     //Waga 1                                                   
	iWeight1State										:INT;						// Stan
	sWeight1State										:STRING;					// Stan
	bWeight1DoWeighting									:BOOL;						// Ważenie
	bWeight1Tare										:BOOL;						// Taruj
	lrWeight1Measured									:LREAL;						// Waga [g]
	lrWeight1Mass										:LREAL;						// Waga masy [g] (na ekranie głównym)
	//Waga 2
	iWeight2State										:INT;						// Stan
	sWeight2State										:STRING;					// Stan
	bWeight2DoWeighting									:BOOL;						// Ważenie
	bWeight2Tare										:BOOL;						// Taruj
	lrWeight2Measured									:LREAL;						// Waga [g]
	lrWeight2Mass										:LREAL;						// Waga masy [g] (na ekranie głównym)
	//Waga 3
	iWeight3State										:INT;						// Stan
	sWeight3State										:STRING;					// Stan
	bWeight3DoWeighting									:BOOL;						// Ważenie
	bWeight3Tare										:BOOL;						// Taruj
	lrWeight3Measured									:LREAL;						// Waga [g]
	lrWeight3Mass										:LREAL;						// Waga masy [g] (na ekranie głównym)
	//Waga 4
	iWeight4State										:INT;						// Stan
	sWeight4State										:STRING;					// Stan
	bWeight4DoWeighting									:BOOL;						// Ważenie
	bWeight4Tare										:BOOL;						// Taruj
	lrWeight4Measured									:LREAL;						// Waga [g]
	lrWeight4Mass										:LREAL;						// Waga masy [g] (na ekranie głównym)
	//Waga 5	
	iWeight5State										:INT;						// Stan
	sWeight5State										:STRING;					// Stan
	bWeight5DoWeighting									:BOOL;						// Ważenie
	bWeight5Tare										:BOOL;						// Taruj
	lrWeight5Measured									:LREAL;						// Waga [g]
	lrWeight5Mass										:LREAL;						// Waga masy [g] (na ekranie głównym)
	//Waga 6
	iWeight6State										:INT;						// Stan
	sWeight6State										:STRING;					// Stan
	bWeight6DoWeighting									:BOOL;						// Ważenie
	bWeight6Tare										:BOOL;						// Taruj
	lrWeight6Measured									:LREAL;						// Waga [g]
	lrWeight6Mass										:LREAL;						// Waga masy [g] (na ekranie głównym)
	                                               
	(*****P05_WeightCorrection******)       
	//Korekcja wag            
	lrDispencer1CorrectionWeight						:LREAL;						// Korekta 1 [ml] (możliwosć edycji)
	lrDispencer2CorrectionWeight						:LREAL;						// Korekta 2 [ml] (możliwosć edycji)
	lrDispencer3CorrectionWeight						:LREAL;						// Korekta 3 [ml] (możliwosć edycji)
	lrDispencer4CorrectionWeight						:LREAL;						// Korekta 4 [ml] (możliwosć edycji)	
	bWeightCorrectionReset								:BOOL;						// Reset

	(*****P06_WickFeeder******)   	
	//Podajnik knotów
	iWickFeederState									: INT;         	// [E_Station] Stan pracy ogólny
	sWickFeederState									: STRING;       // [E_Station] Stan pracy ogólny
	bWickFeederHoming									: BOOL; 		// Wykonanie procedury bazowania podajnika knotów
	bWickFeederHeightSet								: BOOL; 		// Ustawianie wysokoci podnonika podajnika knotów
	lrWickFeederHeightCV								: LREAL; 		// Aktualna wysokoć 
	bWickFeederIgnoreErrors								: BOOL;     	// Ignorowanie błędów dozownika 1 i po wykonaniu pracy ustawienie że wszystko zostało zrobione

	bWickFeederSorterRun								: BOOL; 		// Sortuj
	bWickFeeder1PrepareRun								: BOOL; 		// Pre-Cykl1
	bWickFeeder1Run										: BOOL; 		// Cykl 1
	bWickFeeder2PrepareRun								: BOOL; 		// Pre-Cykl2
	bWickFeeder2Run										: BOOL; 		// Cykl 2

	bWickFeederManualHeightUp							: BOOL; 		// Do góry
	bWickFeederManualHeightDown							: BOOL; 		// Na dół
	bWickFeederManualSorterEngine						: BOOL;			// Sorter
	bWickFeederManualSorterAir							: BOOL;			// Wydmuch
	bWickFeederManualStopper							: BOOL;			// Stoper 
	bWickFeederManualStopper2							: BOOL;			// Stoper2 	
	bWickFeederManualSeparator1							: BOOL;			// Separator tor 1
	bWickFeederManualSeparator2							: BOOL;			// Separator tor 2
	bWickFeederManualSleve1SeparatorActIn				: BOOL;			// Separator tor 1 - rękaw
	bWickFeederManualSleve1SeparatorActOut				: BOOL;			// Separator tor 1 - butelka
	bWickFeederManualSleve2SeparatorActIn				: BOOL;			// Separator tor 2 - rękaw
	bWickFeederManualSleve2SeparatorActOut				: BOOL;			// Separator tor 2 - butelka
	bWickFeederManualHammer1							: BOOL;			//	Wbijak 1 
	bWickFeederManualHammer2							: BOOL;			//	Wbijak 2
	bWickFeederManualFormPositioning					: BOOL;			// Pozycjonowanie formatek

	//Podawanie knotów - przeciąganie	
	iWickFeederDragingStationState						: INT;
	sWickFeederDragingStationState						: STRING;						// Stan 
	bWickFeederDragingStationRun						: BOOL;							// Cykl
	bWickFeederDragingHoming							: BOOL;							// Bazowanie 
	bWickFeederDragingIgnoreError						: BOOL;							// Ignoruj błędy
	bWickFeederDragingManualFork						: BOOL;							// Podnoszenie
	bWickFeederDragingManualLeadBefore1					: BOOL;							// Prowadzenie 1
	bWickFeederDragingManualLeadBefore2					: BOOL;							// Prowadzenie 2
	bWickFeederDragingManualLeft						: BOOL;							// Przód
	bWickFeederDragingManualRight						: BOOL;							// Tył
	bFormsWickFeederDragMoveToEndPosition				: BOOL;                              	
	lrWickFeederDragingStationPositionCV				: LREAL; 

                                             
	(*****P06_LidFeeder******)   	
	//Podajnik platynek
	bLidFeederHoming									: BOOL; 						// Wykonanie procedury bazowania podajnika platynek
	bLidFeederHeightSet									: BOOL; 						// Ustawianie wysokoci podnonika podajnika platynek
	lrLidFeederHeightCV									: LREAL; 						// Aktualna wysokoć stacji podajnika platynek
	bLidFeederIgnoreErrors								: BOOL;     					// Ignorowanie błędów dozownika 1 i po wykonaniu pracy ustawienie że wszystko zostało zrobione
	bLidFeederManualHeightUp							: BOOL; 					 	// Ręczne podnoszenie stacji podajnika platynek
	bLidFeederManualHeightDown							: BOOL; 
	bLidFeederManualFormPositioning						: BOOL;							// Pozycjonowanie formatek pod podawaniem platynek.
	lrFeederDragingStationPositionCV					:LREAL; 

	//Podajnik platynek 1	
	iLidFeeder1State									: INT;         					// [E_Station] Stan pracy ogólny
	sLidFeeder1State									: STRING;         				// [E_Station] Stan pracy ogólny
	bLidFeeder1PrepareRun								: BOOL; 						// Rozkaz pobrania platynki
	bLidFeeder1Run										: BOOL; 						// Rozkaz odłożenia platynki
	lrLidFeeder1HeaterTempCV							: LREAL;						// Temperatura aktualna grzałki podajnika platynek
	bLidFeeder1ManualAct								: BOOL; 						// Ruch ręczny podajnika platynek
	bLidFeeder1ManualAct2								: BOOL; 						// Ruch ręczny siłownika drugiego podajnika platynek
	bLidFeeder1ManualSuckerAct							: BOOL; 						// Ręczne uruchomienie ssawki podajnika platynek
	bLidFeeder1ManualHeaterAct							: BOOL; 						// Ręczne uruchomienie siłownika grzałki podajnika platynek

	//Podajnik platynek 2
	iLidFeeder2State									: INT;         					// [E_Station] Stan pracy ogólny
	sLidFeeder2State									: STRING;         				// [E_Station] Stan pracy ogólny
	bLidFeeder2PrepareRun								: BOOL; 						// Rozkaz pobrania platynki
	bLidFeeder2Run										: BOOL; 						// Rozkaz odłożenia platynki
	lrLidFeeder2HeaterTempCV							: LREAL;						// Temperatura aktualna grzałki podajnika platynek
	bLidFeeder2ManualAct								: BOOL; 						// Ruch ręczny podajnika platynek
	bLidFeeder2ManualAct2								: BOOL; 						// Ruch ręczny siłownika drugiego podajnika platynek
	bLidFeeder2ManualSuckerAct							: BOOL; 						// Ręczne uruchomienie ssawki podajnika platynek
	bLidFeeder2ManualHeaterAct							: BOOL; 						// Ręczne uruchomienie siłownika grzałki podajnika platynek
		
	//Podawanie platynek przeciąganie	
	iLidFeederDragingStationState						: INT;
	sLidFeederDragingStationState						: STRING;					// Stan 
	bLidFeederDragingStationRun							: BOOL;						// Cykl
	bLidFeederDragingHoming								: BOOL;						// Bazowanie 
	bLidFeederDragingIgnoreError						: BOOL;						// Ignoruj błędy
	bLidFeederDragingManualFork							: BOOL;						// Podnoszenie
	bLidFeederDragingManualLeadBefore1					: BOOL;						// Prowadzenie 1
	bLidFeederDragingManualLeadBefore2					: BOOL;						// Prowadzenie 2
	bLidFeederDragingManualLeft							: BOOL;						// Przód
	bLidFeederDragingManualRight						: BOOL;						// Tył
	bFormsLidFeederDragMoveToEndPosition				: BOOL;                              		

	
	//Sprawdzanie platynki
    iLidPuttedCheckState            					: INT;    						// [E_Station] Stan pracy
    sLidPuttedCheckState            					: STRING; 						// Opis stanu pracy
	bLidPuttedCheckRun									: BOOL; 						// Sprawdź
    bLidPuttedCheckHoming           					: BOOL;   						// Bazowanie stacji sprawdzania nasadek
    bLidPuttedCheckHeightSet        					: BOOL;   						// Ustawianie wysokoci stacji sprawdzania nasadek
    bLidPuttedCheckIgnoreErrors     					: BOOL;   						// Ignorowanie błędów stacji sprawdzania nasadek i po wykonaniu pracy ustawienie że wszystko zostało zrobione
    lrLidPuttedCheckHeightCV        					: LREAL;  						// Aktualna wysokoć stacji sprawdzania nasadek
	lrLidPuttedCheckSetPosStepMode						: LREAL;						// Tryb manualny, Ruch podnośnika o zadaną wartość z VIS w trybie krokowym
	bLidPuttedCheckStepMode		 						: BOOL;							// Trzyb manualny, Sterowanie napędem w trybie krokowym.
    bLidPuttedCheckManualHeightUp   					: BOOL;							// Ręczne podnoszenie stacji sprawdzania nasadek
    bLidPuttedCheckManualHeightDown 					: BOOL;							// Reczne opuszczanie stacji sprawdzania nasadek
	bLidPuttedCheckOK									: BOOL;							// Plantyka OK
	AsLidPuttedCheckProgramDescription					: ARRAY [0..20] OF STRING;		// Opis programów kamer, 0 - Opis programu nr 1, 1 - Opis programu nr 2
	
	//Grzałka zasadnicza                                
    bLidSealerHoming									: BOOL;							// Bazowanie stacji zgrzewania zasadniczego
    bLidSealerIgnoreErrors								: BOOL;						    // Ignorowanie błędów Zgrzewarki i po wykonaniu pracy ustawienie że wszystko zostało zrobione
  	lrLidSealerHeightCV									: LREAL;						// Aktualna wysokoć stacji zgrzewania zasadniczego
 	bLidSealerHeightSet									: BOOL;							// Ustawianie wysokości zgrzewarki
    bLidSealerManualHeightUp							: BOOL; 					    // Ręczne podnoszenie stacji grzałki zasadniczej
    bLidSealerManualHeightDown							: BOOL;					    	// Reczne opuszczanie stacji grzałki zasadniczej

	//Grzałka zasadnicza 1                               
	iLidSealer1State									: INT;							// [E_Station] Stan pracy ogólny
	sLidSealer1State									: STRING;						// [E_Station] Stan pracy ogólny
	bLidSealer1Run										: BOOL;							// Rozkaz zgrzania platynki
  	lrLidSealer1HeaterTempCV							: LREAL;						// Temperatura aktualna grzałki zasadniczej
    bLidSealer1ManualAct								: BOOL;							// Ruch ręczny grzałki zasadniczej

	//Stoper
	bLidSealerStoperManualActuator						: BOOL;
	
	//Grzałka zasadnicza 2
	iLidSealer2State									: INT;							// [E_Station] Stan pracy ogólny
	sLidSealer2State									: STRING;						// [E_Station] Stan pracy ogólny
	bLidSealer2Run										: BOOL;							// Rozkaz zgrzania platynki
  	lrLidSealer2HeaterTempCV							: LREAL;						// Temperatura aktualna grzałki zasadniczej
    bLidSealer2ManualAct								: BOOL;							// Ruch ręczny grzałki zasadniczej
		
	//Zgrzanie platynek przeciąganie	
	iLidSealerDragingStationState						: INT;
	sLidSealerDragingStationState						: STRING;					// Stan  
	bLidSealerDragingStationRun							: BOOL;						// Cykl
	bLidSealerDragingHoming								: BOOL;						// Bazowanie
	bLidSealerDragingIgnoreError						: BOOL;						// Ignoruj błędy
	bLidSealerDragingManualFork							: BOOL;						// Podnoszenie
	bLidSealerDragingManualLeadBefore1					: BOOL;						// Prowadzenie 1
	bLidSealerDragingManualLeadBefore2					: BOOL;						// Prowadzenie 2
	bLidSealerDragingManualLeft							: BOOL;						// Przód
	bLidSealerDragingManualRight						: BOOL;						// Tył
	lrSealerDragingStationPositionCV					:LREAL;
	bFormsLidSealerDragMoveToEndPosition			:BOOL;
	
	(*****P08_CapFeeder********)
	// [H] Podajnik nakrętek
	iCapFeederState										:INT;						// [H] Stan
	sCapFeederState										:STRING;					// [H] Stan
    bCapFeederHoming									:BOOL;						// [H] Bazowanie
 	bCapFeederRun										:BOOL; 						// [H] Cykl
	bCapFeederIgnoreErrors								:BOOL;					 	// [H] Ignoruj błędy
	bCapFeederHeightSet									:BOOL;						// [H] Ustaw
	bCapFeederManualHeightUp							:BOOL;						// [H] Do góry
	bCapFeederManualHeightDown							:BOOL;						// [H] Na doł
	bCapFeederManualSorterEngine						:BOOL;						// [H] Silnik
	bCapFeederManualSorterAir							:BOOL;						// [H] Wydmuch
	lrCapFeederHeightCV									:LREAL;						// [H] Aktualna wyskokość 
	bCapFeederManualGate1								:BOOL;						// [H] Szlaban 1
	bCapFeederManualGate2								:BOOL;						// [H] Szlaban 2				                                			

	(*****P08_CapSorter********)	 
	bCapSorterHold										:BOOL; 
	// Przeciąganie formatek pod sorterem nakrętek
	iCapSorterDragState									:INT;						// Stan
	sCapSorterDragState									:STRING;					// Stan
	bCapSorterDragRun									:BOOL;						// Cykl
	bCapSorterDragHoming								:BOOL;						// Bazowanie 
	bCapSorterDragIgnoreError							:BOOL;						// Ignoruj błędy
	bCapSorterDragManualFork							:BOOL;						// Podnosnik
	bCapSorterDragManualLeadBefore1						:BOOL;						// Prowadzenie
	bCapSorterDragManualLeadAfter1						:BOOL;
	bCapSorterDragManualLeft							:BOOL;						// Do przodu
	bCapSorterDragManualRight							:BOOL;						// Do tyłu
	lrCapSorterDragPositionCV							:LREAL;
	bFormsCapSorterDragMoveToEndPosition			:BOOL;
	//Stoper
	bCapSorterStoperManualActuator						: BOOL;

	(*****P09_CapPuttedCheck********) 
	// Sprawdzanie nasadki               			
	iCapPuttedCheckState								:INT;         				// Stan
	sCapPuttedCheckState								:STRING;         			// Stan
    bCapPuttedCheckHoming								:BOOL;					   	// Bazowanie
    bCapPuttedCheckIgnoreErrors							:BOOL := FALSE;				  // Ignoruje błędy
   	lrCapPuttedCheckHeightCV							:LREAL;				 		// Aktualna wysokoć 
    bCapPuttedCheckManualHeightUp						:BOOL; 						// Do góry
    bCapPuttedCheckManualHeightDown						:BOOL;			 			// Na dół
	bCapPuttedCheckHeightSet							:BOOL;						// Ustaw

 	(*****P10_GripperScrewer********)
	//Przeciąganie formatek po zakręcarkami
	iBottleDragingStationState							:INT;						// Stan 
	sBottleDragingStationState							:STRING;					// Stan 
	bBottleDragingStationRun							:BOOL;						// Cykl
	bBottleDragingStationHoming							:BOOL;						// Bazowanie
	bBottleDragingStationIgnoreError					:BOOL;						// Ignoruj błędy
	bBottleDragingStationManualFork1					:BOOL;						// Podnoszenie
	bBottleDragingStationManualLead						:BOOL;						// Prowadzenie
	bBottleDragingStationManualLeft						:BOOL;						// Do przodu
	bBottleDragingStationManualRight					:BOOL;						// Do tyłu
	lrBottleDragingStationPositionCV					:LREAL;
	bFormsScrewersDragMoveToEndPosition				:BOOL;
	
	//Zakręcarki szczękowe 
    bGripperScrewerIgnoreErrors							:BOOL; 						// Ignoruj błędy
  	bGripperScrewerHoming								:BOOL;						// Bazowanie
	bGripperScrewerHeightSet							:BOOL;						// Ustaw
	lrGripperScrewerManualOverride						:LREAL:=100;  				// [H] Prędkość
	AsGripperScrewerTool								:ARRAY [0..10] OF STRING;	// Głowica (1-Opis_narzędzia_nr_1, 2-Opis_narzędzia_nr_2)

	//Zakręcarka 1
	iGripperScrewer1State								:INT;						// Stan
	sGripperScrewer1State								:STRING;					// Stan
	lrGripperScrewer1LiftActPos							:LREAL;	 	  				// Aktualna pozycja
  	bGripperScrewer1Run									:BOOL;						// Cykl
    bGripperScrewer1ManualRight							:BOOL;  					// Obrót w prawo
    bGripperScrewer1ManualLeft							:BOOL;   					// Obrót w lewo
    bGripperScrewer1ManualCatch							:BOOL;  					// Chwyć
  	bGripperScrewer1AdjustTorque						:BOOL;						// [H] Badanie momentu odkręcania
	lrGripperScrewer1AdjustingSetTorque					:LREAL := 1.0;				// [H] Zadany szukany moment otwierania [Nm]
	lrGripperScrewer1TorqueCV							:LREAL;  					// Moment dokręcenia [nM] (po zakręceniu)

	//Zakręcarka 2	
	iGripperScrewer2State								:INT;						// Stan
	sGripperScrewer2State								:STRING;					// Stan
	lrGripperScrewer2LiftActPos							:LREAL;	 	  				// Aktualna pozycja
	bGripperScrewer2Run									:BOOL;                      // Cykl
    bGripperScrewer2ManualRight							:BOOL;  					// Obrót w prawo
    bGripperScrewer2ManualLeft							:BOOL;   					// Obrót w lewo
    bGripperScrewer2ManualCatch							:BOOL;  					// Chwyć
	lrGripperScrewer2TorqueCV							:LREAL;  					// Moment dokręcenia [nM] (po zakręceniu)

	bGripperScrewer1SetPositionOffset					:BOOL;						// Ustaw offset 1
	bGripperScrewer2SetPositionOffset					:BOOL;						// Ustaw offset 2
	
	//Podnośnik zakręcarek
	bGripperScrewerLiftManualHeightUp					:BOOL;  					// Do góry
    bGripperScrewerLiftManualHeightDown						:BOOL;  					// Na dół

	//Chwytak zakrecarki szczękowej
	lrGripperScrewerCatchHeightCV						:LREAL;  					// Aktualna pozycja
	bGripperScrewerCatchHeightSet						:BOOL;						// Ustaw
    bGripperScrewerCatchManualUp						:BOOL;  					// Do góry
    bGripperScrewerCatchManualDown						:BOOL;  					// Na dół

	//Chwytak 1
	iGripperScrewerCatch1State							:INT;						// Stan
	sGripperScrewerCatch1State							:STRING;					// Stan
	bGripperScrewerCatch1ManualActuator					:BOOL;  					// Chwytak
	//chwytak 2
	iGripperScrewerCatch2State							:INT;						// Stan
	sGripperScrewerCatch2State							:STRING;                    // Stan
	bGripperScrewerCatch2ManualActuator					:BOOL;  					// Chwytak
	//Stoper
	bGripperScrewerStoperManualActuator					: BOOL;
		
	
	(*****P11_CapCorrectCheck********) 
	//Sprawdzanie zakręcenia                  			
	iCapCorrectCheckState								:INT;         				// Stan
	sCapCorrectCheckState								:STRING;         			// Stan
    bCapCorrectCheckHoming								:BOOL;					   	// Bazowanie
    bCapCorrectCheckIgnoreErrors						:BOOL;				    	// Ignoruj błędy
   	lrCapCorrectCheckHeightCV							:LREAL;				 		// Aktualna wysokość
    bCapCorrectCheckManualHeightUp						:BOOL; 						// Do góry
    bCapCorrectCheckManualHeightDown					:BOOL;			 			// Na dół
	bCapCorrectCheckHeightSet							:BOOL;						// Ustaw
	AsCapCorrectCheckCameraProgramDescription			:ARRAY [0..10] OF STRING;	// Opis programów kamer, 0 - Opis programu nr 1, 1 - Opis programu nr 2
	bCapCorrectCheckCameraOK							:BOOL;						// Orientacja nasadki OK
                               			
	(*****P13_BottleTransfer********)
	//Przenoszenie butelek
	iBottleTransferState								:INT; 						// Stan
	sBottleTransferState								:STRING;                    // Stan      
	bBottleTransferHoming								:BOOL;  					// Bazowanie 
	bBottleTransferHeightSet 							:BOOL;			 			// Ustaw
	bBottleTransferIgnoreErrors							:BOOL; 						// Ignoruj błedy
	bBottleTransferRun									:BOOL; 						// Cykl Pobierz
    bBottleTransferPlace								:BOOL; 						// Cykl Odłóż
    nBottleTransferPlaceOption							:INT; 					  	// Miejsce odłozenia	(1 - etykieciarka, 2 - odrzut)
	nBottleTransferPickOption							:INT;						// Miejsce pobrania		(1- 1 butelka, 2 - 2 butelki)
	bBottleTransferManualCatch							:BOOL;					 	// Chwytak
    bBottleTransferManualPick							:BOOL; 						// Pobierz 1 but.
	bBottleTransferManualPick2 							:BOOL; 						// Pobierz 2 but.
    bBottleTransferManualPlace1							:BOOL; 						// Odłóż na etykieciarkę
    bBottleTransferManualPlace2							:BOOL; 						// Odłóż na odrzut
    bBottleTransferManualReadyPosition					:BOOL; 						// Gotowość
	bBottleTransferManualStartInkJet					:BOOL; 						// Start InkJet
	bBottleTransferManualStopInkJet						:BOOL; 						// Stop InkJet
	bBottleTransferManualWeight							:BOOL;						// Waga
	bBottleTransferManualEditOffset						:BOOL; 						// Edycja offsetów		
	bBottleTransferAllFormsToLabeler					:BOOL;						// Przekładanie wszystkich na etykieciarkę (opis na głównym: "Przenoszenie wszystkich butelek na etykieciarke") (Umieścić na ekranie głównym)
	bBottleTransferAllFormsToExit						:BOOL;						// Przekadanie wszystkich na odrzut (opis na głównym: "Przenoszenie wszystkich butelek na etykieciarke") (Umieścić na ekranie głównym)
	bBottleTransferLubricationReset						:BOOL;						// Reset smarowania
	aBottleTransferLoadAxis								:ARRAY[0..3] OF INT;		// [H] Aktualne obciążenia osi J1 J2 J3 J4	 
	iBottleTransferLock									:INT;						// Blokowanie przycisków trybu manualnego (b0-1 blokuj 
	bBottleTransferForceWeight							:BOOL;						// Przesuń następne opakowanie na wagę																					// 2#11111111 - nie moge nic  
																					// 2#11111110 - moge pobrać (tylko Pick1 i Pick 2 odblokowane)
																					// 2#11101001 - moge odłożyć, odrzucić i pojechać przed inkjet		
																					// 2#11110111 - moge jechać tylko do gotowości
																					// 2#11110111 - moge jechać tylko do gotowości
																					// 2#11011111 - moge jechać do koniec inkjet
																					// 2#10101101 - moge odłożyć na ety., wrocić przed inkjet
																					// 2#11111110 - moge pobrać

	(*Wersja 2, jeżeli nie uda się odtworzyć widoczności po zmiennej..Lock'	*)																				
	bBottleTransferManualCatchVisibility				:BOOL;					 	// Chwytak - przycisk odblokowany
    bBottleTransferManualPickVisibility					:BOOL; 						// Pobierz 1 but. - przycisk odblokowany
	bBottleTransferManualPick2Visibility 				:BOOL; 						// Pobierz 2 but. - przycisk odblokowany
    bBottleTransferManualPlace1Visibility				:BOOL; 						// Odłóż na etykieciarkę - przycisk odblokowany
    bBottleTransferManualPlace2Visibility				:BOOL; 						// Odłóż na odrzut - przycisk odblokowany
    bBottleTransferManualReadyPositionVisibility		:BOOL; 						// Gotowość - przycisk odblokowany
	bBottleTransferManualStartInkJetVisibility			:BOOL; 						// Start InkJet - przycisk odblokowany
	bBottleTransferManualStopInkJetVisibility			:BOOL; 						// Stop InkJet - przycisk odblokowany

	(*****P13_BottleTransferAfterDrag********)
	//Przeciąganie formatek 
	iBottleTransferAfterDragState						:INT;						// Stan
	sBottleTransferAfterDragState						:STRING;					// Stan
	bBottleTransferAfterDragRun							:BOOL;						// Cykl
	bBottleTransferAfterDragHoming						:BOOL;						// Bazowanie 
	bBottleTransferAfterDragIgnoreError					:BOOL;						// Ignoruj błędy
	bBottleTransferAfterDragManualActuator					:BOOL;						// Podnosnik
	//Stoper,szlaban
	bBottleTransferAfterDragManualStoper				:BOOL;						// Stoper
	bBottleTransferAfterDragManualGate					:BOOL;						// Stoper

	
	(*****P14_BadBottleConyevor********)
	//Transporter odzutu
	iBadBottleConveyorState								:INT; 					 	// Stan
	sBadBottleConveyorState								:STRING; 					// Stan
	nBadBottleConveyorCV								:UDINT; 					// Aktualna prędkość [rpm]
	bBadBottleConveyorManualCmdStart					:BOOL; 						// Start 
	bBadBottleConveyorManualDirection 					:BOOL; 						// Kierunek
	
	(*******P14_TurnTable********)
	
	(********P15_FormTransporters********)
	//Transporter przed dozownikami
	iFormTransporterDispencerState						:INT; 					 	// Stan
	sFormTransporterDispencerState						:STRING; 					// Stan
	nFormTransporterDispencerVelocityCV					:INT;						// Aktualna prędkość
	bFormTransporterDispencerManualCmdStart				:BOOL; 					 	// Start
	//Transporter za dozownikami
	iFormTransporterScrewerState						:INT; 					 	// Stan
	sFormTransporterScrewerState						:STRING; 					// Stan
	nFormTransporterScrewerVelocityCV					:INT;						// Aktualna prędkość
	bFormTransporterScrewerManualCmdStart				:BOOL; 					 	// Start
	//Transporter przed zakręcarką
	iFormTransporterBeforeScrewerState					:INT;						// Stan
	sFormTransporterBeforeScrewerState					:STRING;					// Stan
	nFormTransporterBeforeScrewerVelocityCV				:INT;						// Aktualna prędkość
	bFormTransporterBeforeScrewerManualCmdStart			:BOOL; 						// Start
	//Spowalniacz
	iFormTransporterAfterCapSorterState							:INT;						// Stan pracy spowalniacz formatek
	sFormTransporterAfterCapSorterState							:STRING;					// Stan pracy spowialniacza formatek
	nFormTransporterAfterCapSorterVelocityCV					:INT;						// Aktualna predkosc spowalniacza
	bFormTransporterAfterCapSorterManualCmdStart				:BOOL; 						// Stan pracy spowalniacza formatek
	//Transporter za zakręcarką
	iFormTransporterAfterScreweArState					:INT;						// Stan
	sFormTransporterAfterScrewerState					:STRING;					// Stan
	nFormTransporterAfterScrewerVelocityCV				:INT;						// Aktualna prędkość
	bFormTransporterAfterScrewerManualCmdStart			:BOOL; 						// Start

	(*****P16_LabelMachine********)
	//Etykieciarka
	bLabelMachine1ManualStart 							:BOOL;						// Start
	
	(*****P17_CircularInkJet********)
	//[H] Inkjet obrotowy
	bCircularInkjetRollersManualStart 					:BOOL;						// [H] Rolki
	bCircularInkjetActuatorManualStart 					:BOOL;						// [H] Chwytak
	(*****P17_TurnTables********)
	//Stół odbiorczy
	bExitTurnTable1ManualStart 							:BOOL;						// Start
	bExitTurnTableManualActuator						:BOOL;						// Siłownik stołu odbiorczego
	//Transporter odbiorczy
	bExitConveyorManualStart							:BOOL;						// Transporter
	bExitConveyorGateManualActuator						:BOOL;						// Szlaban transportera odbiorczego
	
	(*****P20_ExhaustFan*****)
	//Wentylator Ex
	iExhaustFanState									:INT;						// Stan
	sExhaustFanState									:STRING;					// Stan
	udiExhaustFanVelocityCV								:UDINT;						// Aktualna prędkość wentylatora
	bExhaustFanManualCmdStart							:BOOL;						// Start
	
	
	bOffPLC			:BOOL;					//sygnał do wyłączenia PLC
	UPPackMLState 	:INT;					//statusy PckML kartoniarki
	EPPackMLState	:INT;					//statusy PckML paletyzatora
	
	//Zmienne do odczytu prądu krokówek
	DCcurrertStepeerScrewers AT%I*:UINT;     
	DCcurrertStepeerDosers AT%I*:UINT;
	
	
	
(********************************************************************************************************************************************)
(********************************************************************************************************************************************)

	(******* Zmienne do receptury*********)

	(*****P00_Recipes***) 
	(*****Receptury****)	
	bChooseRecipe										:BOOL; 						// Wczytaj
	bRecipeLoading 										:BOOL; 						// Trwa wczytywanie
	
	sRecipeNameShow										:WSTRING;		//	P030_Recipes.stActRecipe.stUBL.sRecipeNameShow;		// Nazwa 
	sRecipeDescriptionShow								:WSTRING(1000);	//	P030_Recipes.stActRecipe.stUBL.sRecipeDescriptionShow;		// Nazwa
	sRecipeDispencerDescriptionShow						:WSTRING(250);		
	sRecipeCapsDescriptionShow 							:WSTRING(250);				
	sRecipeFormersDescriptionShow                       :WSTRING(250);
	sRecipeRobotDescriptionShow                         :WSTRING(250);
	sRecipeBottleSorterDescriptionShow                  :WSTRING(250);
	sRecipeCapSorterDescriptionShow                     :WSTRING(250);
	sRecipeCapPutterDescriptionShow                     :WSTRING(250);
                                                                        //
	sRecipeIndexShow									:STRING;		//	P030_Recipes.stActRecipe.stUBL.sRecipeIndexShow;		// Indeks 
	nRecipeIndexShow									:REAL;			//	P030_Recipes.stActRecipe.stUBL.nRecipeIndexShow;		// Indeks 
                                                                        //
	//Parametry opakowania
 	iPackagePuckInsertHeightShow						:INT; 			// Wysokość wkładki w formatce (0-100mm)                
	iPackageMassTypeShow								:INT; 			// Typ masy (0-Woda, 1-Olej, 2-Mydło, 3-Krem itd.)
	iPackageCapTypeShow									:INT; 			// Typ nasadki (0-Fliptop, 1-Pompka/Atomizer, 2-Fliptop z boku, 3-Airless, 4-Deko z boku, 5- Deko
	iPackageCapDiameterShow								:INT;			// Średnica nasadki (5-50mm),
	iPackageHeightShow									:INT;			// Wysokość butelki (50-300mm),
	iPackageCappedHeightShow							:INT;			// Wysokość butelki razem z dokręconą nakrętką i formatką (50-350mm),	
	iPackageNozzleDiameterShow							:INT;			// Srednica wylewki (6-30mm),	
	                                                                        //
	//[H] Praca w trybie wybuchowym                                     //
	bExEnableShow										:BOOL;			//	P030_Recipes.stActRecipe.stUBL.bExEnableShow;		// [H] Tryb EX
	                                                                    //
	// Podajnik butelek  	                                            //
	bBottleFeederEnableShow								:BOOL;   		//	P030_Recipes.stActRecipe.stUBL.bBottleFeederEnableShow							 		// Aktywacja
	iBottleFeederTurntableVelocitySVShow				:UDINT;			//	P030_Recipes.stActRecipe.stUBL.iBottleFeederTurntableVelocitySVShow	// Prędkość stołu
	iBottleFeederBottleSensorDelayShow					:INT;			//	P030_Recipes.stActRecipe.stUBL.iBottleFeederBottleSensorDelayShow		// Opóźnienie wjazdu butelki
	iBottleFeederFormGateDelayShow						:INT;			//	P030_Recipes.stActRecipe.stUBL.iBottleFeederFormGateDelayShow			// Czas otwarcia szlabanu formatek
	iBottleFeederAllowFormDelayShow						:INT;			//	P030_Recipes.stActRecipe.stUBL.iBottleFeederAllowFormDelayShow			// Czas po którym formatka zostaje wypuszczona bez butelki
                                                                        //
	// Podajnik opakowań	                                            //
	bPucksInserterEnableShow							:BOOL;   		//	P030_Recipes.stActRecipe.stUBL.bPucksInserterEnableShow						// Aktywacja
	iPucksInserterTurntableVelocitySVShow				:UDINT;			//	P030_Recipes.stActRecipe.stUBL.iPucksInserterTurntableVelocitySVShow			// Prędkość stołu
	iPucksInserterConveyorVelocitySVShow				:UDINT;			//	P030_Recipes.stActRecipe.stUBL.iPucksInserterConveyorVelocitySVShow			// Prędkość transportera
	iPucksInserterBottleSensorDelayShow					:INT;			//	P030_Recipes.stActRecipe.stUBL.iPucksInserterBottleSensorDelayShow				// Opóźnienie wjazdu butelki
	iPucksInserterFormGateDelayShow						:INT;			//	P030_Recipes.stActRecipe.stUBL.iPucksInserterFormGateDelayShow					// Czas otwarcia szlabanu formatek
	iPucksInserterAllowFormDelayShow					:INT;			//	P030_Recipes.stActRecipe.stUBL.iPucksInserterAllowFormDelayShow				// Czas po którym formatka zostaje wypuszczona bez butelki
	lrPucksInserterWheelOffsetShow						:LREAL;			//	P030_Recipes.stActRecipe.stUBL.lrPucksInserterWheelOffsetShow					// Offset karuzeli +-10 st.
	lrPucksInserterWheelAccelerationShow				:LREAL;			//	P030_Recipes.stActRecipe.stUBL.lrPucksInserterWheelAccelerationShow			// Przyspieszenie 
	lrPucksInserterWheelVelocityShow					:LREAL;			//	P030_Recipes.stActRecipe.stUBL.lrPucksInserterWheelVelocityShow				// Prędkość 
	lrPucksInserterHammerHeightSVShow					:LREAL;  		//	P030_Recipes.stActRecipe.stUBL.lrPucksInserterHammerHeightSVShow				// Zadana wysokość
	                                                                    //                                                                                    									
	//Vasyl 27.05 Stół podający butelki                                 //                                               									
	udiPucksInserterPushTableVelocityShow				:UDINT;			//	P030_Recipes.stActRecipe.stUBL.udiPucksInserterPushTableVelocityShow			 									
	iPucksInserterPushTableRollersVelocityShow			:INT;           //  P030_Recipes.stActRecipe.stUBL.iPucksInserterPushTableRollersVelocityShow		 									
	udiPucksInserterPushTableActuatorPUSHDelayShow		:UDINT;         //  P030_Recipes.stActRecipe.stUBL.udiPucksInserterPushTableActuatorPUSHDelayShow	 									
	udiPucksInserterPushTableActuatorPULLDelayShow		:UDINT;         //  P030_Recipes.stActRecipe.stUBL.udiPucksInserterPushTableActuatorPULLDelayShow	 									
	bPucksInserterPushTableActuatorEnableShow			:BOOL;          //  P030_Recipes.stActRecipe.stUBL.bPucksInserterPushTableActuatorEnableShow		 									
	bPucksInserterPushTableRollerEnableShow				:BOOL;          //  P030_Recipes.stActRecipe.stUBL.bPucksInserterPushTableRollerEnableShow			 									
	bPucksInserterPushTableEnableShow					:BOOL;          //  P030_Recipes.stActRecipe.stUBL.bPucksInserterPushTableEnableShow				 	
	udiPucksInserterPushTableOFFDelayShow				:UDINT;			//	P030_Recipes.stActRecipe.stUBL.udiPucksInserterPushTableOFFDelayShow					
	                                                                    //
	                                                                    //
	//Sorter butelek                                                    //
	//Parametry receptur z innego sterownika                            //
	                                                                    //
	//[H] Parametry szlabanów                                           //
	bGateBeforeDispencersEnableShow						:BOOL;			//	P030_Recipes.stActRecipe.stUBL.bGateBeforeDispencersEnableShow									// [H] Aktywacja
	nGateBeforeDispencersTimeFormInsertingShow			:UINT;			//	P030_Recipes.stActRecipe.stUBL.nGateBeforeDispencersTimeFormInsertingShow						// [H] Czas wyjazdu formatki	
	bGateAfterWeightEnableShow							:BOOL;			//	P030_Recipes.stActRecipe.stUBL.bGateAfterWeightEnableShow										// [H] Aktywacja
	nGateAfterWeightTimeFormInsertingShow				:UINT;			//	P030_Recipes.stActRecipe.stUBL.nGateAfterWeightTimeFormInsertingShow							// [H] Czas wyjazdu formatki
	bGateRobotEnableShow								:BOOL;			//	P030_Recipes.stActRecipe.stUBL.bGateRobotEnableShow											// [H] Aktywacja
	nGateRobotTimeFormInsertingShow						:UINT;			//	P030_Recipes.stActRecipe.stUBL.nGateRobotTimeFormInsertingShow									// [H] Czas przejazdu formatki
                                                                        //                                        										
	//Przeciaganie formatek pod dozownikami	lewe                        //                                        										
	bFormsDragingLeftEnableShow							:BOOL;			//	P030_Recipes.stActRecipe.stUBL.bFormsDragingLeftEnableShow								// Aktywacja
	lrFormsDragingLeftVelocityShow						:LREAL; 		//	P030_Recipes.stActRecipe.stUBL.lrFormsDragingLeftVelocityShow							// Prędkość [mm/s] (100-1000)
 	lrFormsDragingLeftAccelerationShow					:LREAL;			//	P030_Recipes.stActRecipe.stUBL.lrFormsDragingLeftAccelerationShow					// Przyspieszenie [mm/s2] (100-10000)
	lrFormsDragingLeftDecelerationShow					:LREAL;			//	P030_Recipes.stActRecipe.stUBL.lrFormsDragingLeftDecelerationShow					// Hamowanie [mm/s2] (100-10000)
	//Przeciaganie formatek pod dozownikami	prawe	                    //                                        										
	bFormsDragingRightEnableShow						:BOOL;			//	P030_Recipes.stActRecipe.stUBL.bFormsDragingRightEnableShow							// Aktywacja
	lrFormsDragingRightVelocityShow						:LREAL; 		//	P030_Recipes.stActRecipe.stUBL.lrFormsDragingRightVelocityShow							// Prędkość [mm/s] (100-1000)   
 	lrFormsDragingRightAccelerationShow					:LREAL;			//	P030_Recipes.stActRecipe.stUBL.lrFormsDragingRightAccelerationShow						// Przyspieszenie [mm/s2] (100-1
	lrFormsDragingRightDecelerationShow					:LREAL;			//	P030_Recipes.stActRecipe.stUBL.lrFormsDragingRightDecelerationShow						// Hamowanie [mm/s2] (100-10000)
	                                                                    //                                        												
	//Dozowniki                                                         //                                        												
	bDosingTwoPhasesShow								:BOOL;			//	P030_Recipes.stActRecipe.stUBL.bDosingTwoPhasesShow																			// Dozowanie dwu-fazowe
    lrDispencersLifterReadyPositionShow					:LREAL;			//	P030_Recipes.stActRecipe.stUBL.lrDispencersLifterReadyPositionShow																// Pozycja gototości 
	uiDispencerStartDosingDelayShow						:UINT;			//	P030_Recipes.stActRecipe.stUBL.uiDispencerStartDosingDelayShow																	// Zwłoka rozpoczęcia dozowania
	bDispencer1EnableShow								:BOOL; 			//	P030_Recipes.stActRecipe.stUBL.bDispencer1EnableShow								// Aktywacja dozownika 1                                                        				
	bDispencer2EnableShow								:BOOL; 			//	P030_Recipes.stActRecipe.stUBL.bDispencer2EnableShow								// Aktywacja dozownika 2 
	bDispencer3EnableShow								:BOOL; 			//	P030_Recipes.stActRecipe.stUBL.bDispencer3EnableShow								// Aktywacja dozownika 3  
	bDispencer4EnableShow								:BOOL; 			//	P030_Recipes.stActRecipe.stUBL.bDispencer4EnableShow								// Aktywacja dozownika 4  
	                                                                    //
	//Dozownik 12 (druga faza)                                       	//			
	lrDispencer1DoseVolumeShow							:LREAL:=300; 	//	P030_Recipes.stActRecipe.stUBL.lrDispencer1DoseVolumeShow						// Objętość do wydozowania [ml]
	lrDispencer1Phase1VolumeShow						:LREAL:=100;	//	P030_Recipes.stActRecipe.stUBL.lrDispencer1Phase1VolumeShow					// Objętość fazy początkowej [ml]
	lrDispencer1Phase2VolumeShow						:LREAL:=200;	//	P030_Recipes.stActRecipe.stUBL.lrDispencer1Phase2VolumeShow					// Objętość fazy końcowej [ml]
	lrDispencer1Phase1VelocityShow						:LREAL:=500;	//	P030_Recipes.stActRecipe.stUBL.lrDispencer1Phase1VelocityShow					// Prędkość fazy początkowej [ml/s]
	lrDispencer1Phase2VelocityShow						:LREAL:=500;	//	P030_Recipes.stActRecipe.stUBL.lrDispencer1Phase2VelocityShow					// Prędkość fazy dozowania [ml/s]
	lrDispencer1Phase3VelocityShow						:LREAL:=500;	//	P030_Recipes.stActRecipe.stUBL.lrDispencer1Phase3VelocityShow					// Prędkość fazy koncowej [ml/s]
	lrDispencer1SuckVelocityShow						:LREAL:=500;	//	P030_Recipes.stActRecipe.stUBL.lrDispencer1SuckVelocityShow					// Prędkość zasysania masy [ml/s2]
	lrDispencer1Phase1AccelerationShow					:LREAL:=3000;	//	P030_Recipes.stActRecipe.stUBL.lrDispencer1Phase1AccelerationShow				// Przyśpieszenie fazy początkowej [ml/s2]
	lrDispencer1Phase2AccelerationShow					:LREAL:=3000;	//	P030_Recipes.stActRecipe.stUBL.lrDispencer1Phase2AccelerationShow				// Przyśpieszenie fazy dozowania [ml/s2]
	lrDispencer1Phase3AccelerationShow					:LREAL:=3000;	//	P030_Recipes.stActRecipe.stUBL.lrDispencer1Phase3AccelerationShow				// Przyśpieszenie fazy końcowej [ml/s2]
	lrDispencer1SuckAccelerationShow					:LREAL:=3000;	//	P030_Recipes.stActRecipe.stUBL.lrDispencer1SuckAccelerationShow				// Przyśpieszenie zasysania masy [ml/s2]
	lrDispencer1Phase1DecelerationShow					:LREAL:=3000;	//	P030_Recipes.stActRecipe.stUBL.lrDispencer1Phase1DecelerationShow				// Dynamika zwalniania w fazie początkowej
	lrDispencer1Phase2DecelerationShow					:LREAL:=3000;	//	P030_Recipes.stActRecipe.stUBL.lrDispencer1Phase2DecelerationShow				// Dynamika zwalniania dozowania
	lrDispencer1Phase3DecelerationShow					:LREAL:=3000;	//	P030_Recipes.stActRecipe.stUBL.lrDispencer1Phase3DecelerationShow				// Dynamika zwalniania fazy końcowej
	udiDispencer1DosingDoneDelayTimeShow				:UDINT:=0; 		//	P030_Recipes.stActRecipe.stUBL.udiDispencer1DosingDoneDelayTimeShow			// Zwłoka po wydozowaniu
	lrDispencer1SuckValveOpenVolumeShow					:LREAL:=0;		//	P030_Recipes.stActRecipe.stUBL.lrDispencer1SuckValveOpenVolumeShow				// Objętość przy której otwiera się zawór ssania [3] 
	lrDispencer1SuckValveOpenTimeDelayShow				:LREAL:=0;		//	P030_Recipes.stActRecipe.stUBL.lrDispencer1SuckValveOpenTimeDelayShow			// Zwłoka rozpoczęcia ssania po tłoczeniu [ms] [3]
	lrDispencer1SuckValveCloseVolumeShow				:LREAL:=0;		//	P030_Recipes.stActRecipe.stUBL.lrDispencer1SuckValveCloseVolumeShow			// [H] Objętość zamknięcia zaworu ssania od końca ssania [4]
	lrDispencer1SuckValveCloseTimeDelayShow				:LREAL:=0;		//	P030_Recipes.stActRecipe.stUBL.lrDispencer1SuckValveCloseTimeDelayShow			// Zwłoka zamknięcia zaworu ssącego [ms] [4] 
	lrDispencer1DoseValveOpenVolumeShow					:LREAL:=0;		//	P030_Recipes.stActRecipe.stUBL.lrDispencer1DoseValveOpenVolumeShow				// [H] Objętość przy której otwiera się zawór tłoczenia [ml] [1]
	lrDispencer1DoseValveOpenTimeAccShow				:LREAL:=0;		//	P030_Recipes.stActRecipe.stUBL.lrDispencer1DoseValveOpenTimeAccShow			// Wyprzedzenie otwarcia zaworu tłoczenia [1] [ms]
	lrDispencer1DoseValveCloseVolumeShow				:LREAL:=0;		//	P030_Recipes.stActRecipe.stUBL.lrDispencer1DoseValveCloseVolumeShow			// Pozostała objętość dozy - zamknięcie zaworu tłoczenia [ml] [2]
	lrDispencer1DoseValveCloseTimeDecShow				:LREAL:=0;		//	P030_Recipes.stActRecipe.stUBL.lrDispencer1DoseValveCloseTimeDecShow			// Zwłoka zamkniecia zaworu tłoczenia [2] [ms]
	lrDispencer1DoseSuckingVolumeShow					:LREAL:=0;		//	P030_Recipes.stActRecipe.stUBL.lrDispencer1DoseSuckingVolumeShow				// Ilość dozy do posysenia [ml]	[5] [Podsysanie] 
	lrDispencer1DoseSuckingTimeDelayShow				:LREAL:=0;		//	P030_Recipes.stActRecipe.stUBL.lrDispencer1DoseSuckingTimeDelayShow			// Opóźnienie podsysania [ms] [6] [Podsysanie] 
	bDispencer1DoseSuckingShow							:BOOL;			//	P030_Recipes.stActRecipe.stUBL.bDispencer1DoseSuckingShow						// Aktywacja podsysania
	bDispencer1LiftSynchroPh1Show						:BOOL;			//	P030_Recipes.stActRecipe.stUBL.bDispencer1LiftSynchroPh1Show					// Synchronizacja z podnosnikiem w fazie początkowej
	bDispencer1LiftSynchroPh2Show						:BOOL; 			//	P030_Recipes.stActRecipe.stUBL.bDispencer1LiftSynchroPh2Show					// Synchronizacja z podnosnikiem w fazie dozowania
	bDispencer1LiftSynchroPh3Show						:BOOL; 			//	P030_Recipes.stActRecipe.stUBL.bDispencer1LiftSynchroPh3Show					// Synchronizacja z podnosnikiem w fazie końcowej
	lrDispencer1LifterStartDosePositionShow				:LREAL:=20;		//	P030_Recipes.stActRecipe.stUBL.lrDispencer1LifterStartDosePositionShow			// Pozycja rozpoczęcia dozowania
	lrDispencer1LifterStopDosePositionShow				:LREAL:=60;		//	P030_Recipes.stActRecipe.stUBL.lrDispencer1LifterStopDosePositionShow			// Pozycja zakończenia dozowania
	lrDispencer1LifterVelocityShow						:LREAL:=100;	//	P030_Recipes.stActRecipe.stUBL.lrDispencer1LifterVelocityShow					// [H] Prędkość podnośnika 
	lrDispencer1LifterAccelerationShow					:LREAL:=2;		//	P030_Recipes.stActRecipe.stUBL.lrDispencer1LifterAccelerationShow				// [H] Przyspieszenie podnośnika
	lrDispencer1LifterDecelerationShow					:LREAL:=2;		//	P030_Recipes.stActRecipe.stUBL.lrDispencer1LifterDecelerationShow				// [H] Zwalnianie podnośnika
                                                                        //
	//Dozowniki 34 (pierwsza faza)                                      //       				
    lrDispencer2DoseVolumeShow							:LREAL:=300; 	//	P030_Recipes.stActRecipe.stUBL.lrDispencer2DoseVolumeShow						// Objętość do wydozowania                                           
	lrDispencer2Phase1VolumeShow						:LREAL:=100;	//	P030_Recipes.stActRecipe.stUBL.lrDispencer2Phase1VolumeShow					// Objętość fazy początkowej                                         
	lrDispencer2Phase2VolumeShow						:LREAL:=200;	//	P030_Recipes.stActRecipe.stUBL.lrDispencer2Phase2VolumeShow					// Objętość fazy końcowej                                            
	lrDispencer2Phase1VelocityShow						:LREAL:=500;	//	P030_Recipes.stActRecipe.stUBL.lrDispencer2Phase1VelocityShow					// Prędkość fazy początkowej                                         
	lrDispencer2Phase2VelocityShow						:LREAL:=500;	//	P030_Recipes.stActRecipe.stUBL.lrDispencer2Phase2VelocityShow					// Prędkość fazy dozowania                                           
	lrDispencer2Phase3VelocityShow						:LREAL:=500;	//	P030_Recipes.stActRecipe.stUBL.lrDispencer2Phase3VelocityShow					// Prędkość fazy koncowej                                            
	lrDispencer2SuckVelocityShow						:LREAL:=500;	//	P030_Recipes.stActRecipe.stUBL.lrDispencer2SuckVelocityShow					// Prędkość zasysania masy                                           
	lrDispencer2Phase1AccelerationShow					:LREAL:=3000;	//	P030_Recipes.stActRecipe.stUBL.lrDispencer2Phase1AccelerationShow				// Przyspieszenie fazy początkowej                                   
	lrDispencer2Phase2AccelerationShow					:LREAL:=3000;	//	P030_Recipes.stActRecipe.stUBL.lrDispencer2Phase2AccelerationShow				// Przyspieszenie fazy dozowania                                     
	lrDispencer2Phase3AccelerationShow					:LREAL:=3000;	//	P030_Recipes.stActRecipe.stUBL.lrDispencer2Phase3AccelerationShow				// Przyspieszenie fazy końcowej                                      
	lrDispencer2SuckAccelerationShow					:LREAL:=3000;	//	P030_Recipes.stActRecipe.stUBL.lrDispencer2SuckAccelerationShow				// Przyspieszenie zasysania masy                                     
	lrDispencer2Phase1DecelerationShow					:LREAL:=3000;	//	P030_Recipes.stActRecipe.stUBL.lrDispencer2Phase1DecelerationShow				// Dynamika zwalniania w fazie początkowej                           
	lrDispencer2Phase2DecelerationShow					:LREAL:=3000;	//	P030_Recipes.stActRecipe.stUBL.lrDispencer2Phase2DecelerationShow				// Dynamika zwalniania dozowania                                     
	lrDispencer2Phase3DecelerationShow					:LREAL:=3000;	//	P030_Recipes.stActRecipe.stUBL.lrDispencer2Phase3DecelerationShow				// Dynamika zwalniania fazy końcowej                                 
	udiDispencer2DosingDoneDelayTimeShow				:UDINT:=0; 		//	P030_Recipes.stActRecipe.stUBL.udiDispencer2DosingDoneDelayTimeShow			// Zwłoka po wydozowaniu                                             
	lrDispencer2SuckValveOpenVolumeShow					:LREAL:=0;		//	P030_Recipes.stActRecipe.stUBL.lrDispencer2SuckValveOpenVolumeShow				// Objętość przy której otwiera się zawór ssania [3]                 
	lrDispencer2SuckValveOpenTimeDelayShow				:LREAL:=0;		//	P030_Recipes.stActRecipe.stUBL.lrDispencer2SuckValveOpenTimeDelayShow			// Zwłoka rozpoczęcia ssania po tłoczeniu [ms] [3]                   
	lrDispencer2SuckValveCloseVolumeShow				:LREAL:=0;		//	P030_Recipes.stActRecipe.stUBL.lrDispencer2SuckValveCloseVolumeShow			// [H] Objętość zamknięcia zaworu ssania od końca ssania [4]    
	lrDispencer2SuckValveCloseTimeDelayShow				:LREAL:=0;		//	P030_Recipes.stActRecipe.stUBL.lrDispencer2SuckValveCloseTimeDelayShow			// Zwłoka zamknięcia zaworu ssącego [ms] [4]                         
	lrDispencer2DoseValveOpenVolumeShow					:LREAL:=0;		//	P030_Recipes.stActRecipe.stUBL.lrDispencer2DoseValveOpenVolumeShow				// [H] Objętość przy której otwiera się zawór tłoczenia [ml] [1]
	lrDispencer2DoseValveOpenTimeAccShow				:LREAL:=0;		//	P030_Recipes.stActRecipe.stUBL.lrDispencer2DoseValveOpenTimeAccShow			// Wyprzedzenie otwarcia zaworu tłoczenia [1] [ms]                   
	lrDispencer2DoseValveCloseVolumeShow				:LREAL:=0;		//	P030_Recipes.stActRecipe.stUBL.lrDispencer2DoseValveCloseVolumeShow			// Pozostała objętość dozy - zamknięcie zaworu tłoczenia [ml] [2]    
	lrDispencer2DoseValveCloseTimeDecShow				:LREAL:=0;		//	P030_Recipes.stActRecipe.stUBL.lrDispencer2DoseValveCloseTimeDecShow			// Zwłoka zamkniecia zaworu tłoczenia [2] [ms]                       
	lrDispencer2DoseSuckingVolumeShow					:LREAL:=0;		//	P030_Recipes.stActRecipe.stUBL.lrDispencer2DoseSuckingVolumeShow				// Ilość dozy do posysenia [ml]	[5] [Podsysanie]                     
	lrDispencer2DoseSuckingTimeDelayShow				:LREAL:=0;		//	P030_Recipes.stActRecipe.stUBL.lrDispencer2DoseSuckingTimeDelayShow			// Opóźnienie podsysania [ms] [6] [Podsysanie]                       
	bDispencer2DoseSuckingShow							:BOOL;			//	P030_Recipes.stActRecipe.stUBL.bDispencer2DoseSuckingShow						// Aktywacja podsysania                                              
	bDispencer2LiftSynchroPh1Show						:BOOL;			//	P030_Recipes.stActRecipe.stUBL.bDispencer2LiftSynchroPh1Show					// Synchronizacja z podnosnikiem w fazie początkowej                 
	bDispencer2LiftSynchroPh2Show						:BOOL; 			//	P030_Recipes.stActRecipe.stUBL.bDispencer2LiftSynchroPh2Show					// Synchronizacja z podnosnikiem w fazie dozowania                   
	bDispencer2LiftSynchroPh3Show						:BOOL; 			//	P030_Recipes.stActRecipe.stUBL.bDispencer2LiftSynchroPh3Show					// Synchronizacja z podnosnikiem w fazie końcowej                    
	lrDispencer2LifterStartDosePositionShow				:LREAL:=20;		//	P030_Recipes.stActRecipe.stUBL.lrDispencer2LifterStartDosePositionShow			// Pozycja rozpoczęcia dozowania                                     
	lrDispencer2LifterStopDosePositionShow				:LREAL:=60;		//	P030_Recipes.stActRecipe.stUBL.lrDispencer2LifterStopDosePositionShow			// Pozycja zakończenia dozowania                                     
	lrDispencer2LifterVelocityShow						:LREAL:=100;	//	P030_Recipes.stActRecipe.stUBL.lrDispencer2LifterVelocityShow					// [H] Prędkość podnośnika                                      
	lrDispencer2LifterAccelerationShow					:LREAL:=2;		//	P030_Recipes.stActRecipe.stUBL.lrDispencer2LifterAccelerationShow				// [H] Przyspieszenie podnośnika                                
	lrDispencer2LifterDecelerationShow					:LREAL:=2;		//	P030_Recipes.stActRecipe.stUBL.lrDispencer2LifterDecelerationShow				// [H] Zwalnianie podnośnika                                    
                                                            		    //
	//Chwytak dozowników 1234                                           //
	bDispencersCatchEnableShow	      					:BOOL;			//	P030_Recipes.stActRecipe.stUBL.bDispencersCatchEnableShow	      			// [H] Aktywacja    
 	bDispencersCatchMaxPressureShow	      				:BOOL;			//	P030_Recipes.stActRecipe.stUBL.bDispencersCatchMaxPressureShow	    		// Zwiększona siła chwytania            		
	lrDispencersCatchHeightSVShow						:LREAL:=86;  	//	P030_Recipes.stActRecipe.stUBL.lrDispencersCatchHeightSVShow				// Pozycja chwytaka
 	//Kalibracja chwytaków 1234                                         //
    lrDispencersCatch1ClosedValueShow                   :LREAL;         //  P030_Recipes.stActRecipe.stUBL.lrDispencersCatch1ClosedValueShow        // Chwytak 1 | wartość kalibracji zamkniętego chwytaka
    lrDispencersCatch1OpenValueShow                     :LREAL;         //  P030_Recipes.stActRecipe.stUBL.lrDispencersCatch1OpenValueShow           // Chwytak 1 | wartość kalibracji otwartego chwytaka
    lrDispencersCatch2ClosedValueShow                   :LREAL;         //  P030_Recipes.stActRecipe.stUBL.lrDispencersCatch2ClosedValueShow         // Chwytak 2 | wartość kalibracji zamkniętego chwytaka
    lrDispencersCatch2OpenValueShow                     :LREAL;         //  P030_Recipes.stActRecipe.stUBL.lrDispencersCatch2OpenValueShow           // Chwytak 2 | wartość kalibracji otwartego chwytaka
    lrDispencersCatch3ClosedValueShow                	:LREAL;         //  P030_Recipes.stActRecipe.stUBL.lrDispencersCatch3ClosedValueShow         // Chwytak 3 | wartość kalibracji zamkniętego chwytaka
    lrDispencersCatch3OpenValueShow                     :LREAL;         //  P030_Recipes.stActRecipe.stUBL.lrDispencersCatch3OpenValueShow           // Chwytak 3 | wartość kalibracji otwartego chwytaka
    lrDispencersCatch4ClosedValueShow                   :LREAL;         //  P030_Recipes.stActRecipe.stUBL.lrDispencersCatch4ClosedValueShow         // Chwytak 4 | wartość kalibracji zamkniętego chwytaka
    lrDispencersCatch4OpenValueShow                     :LREAL;         //  P030_Recipes.stActRecipe.stUBL.lrDispencersCatch4OpenValueShow          // Chwytak 4 | wartość kalibracji otwartego chwytaka
    lrDispencersCatchToleranceShow                      :LREAL;         //  P030_Recipes.stActRecipe.stUBL.lrDispencersCatchToleranceShow            // Tolerancja chwytaka [0-100%]      
                                              		                    //
	//Zbiorniki                                                         //
	bTank1MixerEnableShow								:BOOL;	   		//	P030_Recipes.stActRecipe.stUBL.bTank1MixerEnableShow				// Mieszadło
	bTankHeatingEnableShow								:BOOL;   		//	P030_Recipes.stActRecipe.stUBL.bTankHeatingEnableShow				// Grzanie                                     		
	iTankHeatingTempSVShow								:INT;			//	P030_Recipes.stActRecipe.stUBL.iTankHeatingTempSVShow				// Temperatura
	bTank1PressureEnableShow							:BOOL;  		//	P030_Recipes.stActRecipe.stUBL.bTank1PressureEnableShow			// Ciśnienie                                   		
	bTank1SupplyPumpEnableShow							:BOOL;  		//	P030_Recipes.stActRecipe.stUBL.bTank1SupplyPumpEnableShow			// Aktywacja pompy 1
	bTank2SupplyPumpEnableShow							:BOOL;  		//	P030_Recipes.stActRecipe.stUBL.bTank2SupplyPumpEnableShow			// Aktywacja pompy 2
	uTank1LevelSetpointShow								:UINT;			//	P030_Recipes.stActRecipe.stUBL.uTank1LevelSetpointShow				// [H] Wartość zadana masy do czujnika poziomu w zbiorniku nr 1
	uTank2LevelSetpointShow								:UINT;			//	P030_Recipes.stActRecipe.stUBL.uTank2LevelSetpointShow				// [H] Wartość zadana masy do czujnika poziomu w zbiorniku nr 2
	bTank1LevelSignalInvertShow							:BOOL;			//	P030_Recipes.stActRecipe.stUBL.bTank1LevelSignalInvertShow			// [H] Odwróć sygnał z czujnika zbiornika pierwszego
	bTank2LevelSignalInvertShow							:BOOL;			//	P030_Recipes.stActRecipe.stUBL.bTank2LevelSignalInvertShow			// [H] Odwróć sygnał z czujnika zbionirka drugiego
 	//Zbiorniki-dodatkowe
	bTankRainbowModeShow								:BOOL;			// Tryb 4 zbiorników                 

                          			                //
	//Waga                                           					//	
	bWeight1EnableShow									:BOOL;			//	P030_Recipes.stActRecipe.stUBL.bWeight1EnableShow					// Aktywacja
	lrWeightMassSVShow 									:LREAL;			//	P030_Recipes.stActRecipe.stUBL.lrWeightMassSVShow 					// Waga zadana 
	iWeight1ActuatorUpDelayShow							: INT;			//	P030_Recipes.stActRecipe.stUBL.iWeight1ActuatorUpDelayShow		// Opóźnienie podnoszenia wagi 1
	iWeight2ActuatorUpDelayShow							: INT;			//	P030_Recipes.stActRecipe.stUBL.iWeight2ActuatorUpDelayShow		// Opóźnienie podnoszenia wagi 2
	iWeight3ActuatorUpDelayShow							: INT;			//	P030_Recipes.stActRecipe.stUBL.iWeight3ActuatorUpDelayShow		// Opóźnienie podnoszenia wagi 3
	iWeight4ActuatorUpDelayShow							: INT;			//	P030_Recipes.stActRecipe.stUBL.iWeight4ActuatorUpDelayShow		// Opóźnienie podnoszenia wagi 4
	iWeight5ActuatorUpDelayShow							: INT;			//	P030_Recipes.stActRecipe.stUBL.iWeight5ActuatorUpDelayShow		// Opóźnienie podnoszenia wagi 5 
	iWeight6ActuatorUpDelayShow							: INT;			//	P030_Recipes.stActRecipe.stUBL.iWeight6ActuatorUpDelayShow		// Opóźnienie podnoszenia wagi 6
	                                                                    //
	//Korekcja wagi                                     			    //
	lrFormWeightShow 									:LREAL;			//	P030_Recipes.stActRecipe.stUBL.lrFormWeightShow 								// [H] Waga formatki
	lrMass1DensityShow									:LREAL;			//	P030_Recipes.stActRecipe.stUBL.lrMass1DensityShow								// [H] Gęstoć masy pierwszej fazy [g/ml]
	lrMass2DensityShow									:LREAL;			//	P030_Recipes.stActRecipe.stUBL.lrMass2DensityShow								// [H] Gęstoć masy drugiej fazy [g/ml]
	lrCupWeightShow										:LREAL;			//	P030_Recipes.stActRecipe.stUBL.lrCupWeightShow									// Waga opakowania (z platynką, zależnie od opakowania) [g]
	lrWholePackageWeightShow							:LREAL;			//	P030_Recipes.stActRecipe.stUBL.lrWholePackageWeightShow						// [H] Waga całego opakowania bez masy (kubeczek,platynka,nakrętka) [g]
	lrWeight1MeasurmentCorrectionShow					:LREAL;			//	P030_Recipes.stActRecipe.stUBL.lrWeight1MeasurmentCorrectionShow				// [H] Korekta wagi zmierzonej [g] , różnica pomiedzy wskazaniami wagi zewnętrznej a linią
	bDispencer1WeightCorrectionEnableShow				:BOOL;			//	P030_Recipes.stActRecipe.stUBL.bDispencer1WeightCorrectionEnableShow			// Aktywacja korekcji 1
	bDispencer2WeightCorrectionEnableShow				:BOOL;			//	P030_Recipes.stActRecipe.stUBL.bDispencer2WeightCorrectionEnableShow			// Aktywacja korekcji 2
	bDispencer3WeightCorrectionEnableShow				:BOOL;			//	P030_Recipes.stActRecipe.stUBL.bDispencer3WeightCorrectionEnableShow			// Aktywacja korekcji 3
	bDispencer4WeightCorrectionEnableShow				:BOOL;			//	P030_Recipes.stActRecipe.stUBL.bDispencer4WeightCorrectionEnableShow			// Aktywacja korekcji 4	
	lrWeightUpperToleranceShow							:LREAL;			//	P030_Recipes.stActRecipe.stUBL.lrWeightUpperToleranceShow						// Górny zakres wagi [g]
	lrWeightLowerToleranceShow							:LREAL;			//	P030_Recipes.stActRecipe.stUBL.lrWeightLowerToleranceShow						// Dolny zakres wagi [g]
    iWeightCorrectionNumberOfSamplesShow				:UINT:=2;		//	P030_Recipes.stActRecipe.stUBL.iWeightCorrectionNumberOfSamplesShow			// Ilość próbek korekcji [x] (1-20)

 	//Podajnik knotów                                               
	bWickFeederEnableShow								:BOOL;			//	P030_Recipes.stActRecipe.stUBL.bLidFeederEnableShow				// Zezwolenie na pracę podajnika platynek 
	lrWickFeederHeightPosSVShow							:LREAL;			//	P030_Recipes.stActRecipe.stUBL.lrLidFeederHeightPosSVShow			// Wysokość na której ma znajdować się podajnik platynek
	iWickFeederSorterTimeDelayOnShow					: INT;
	iWickFeederSorterTimeDelayOffShow					: INT;
	iWickFeederSorterTimeToEmptySleeveErrorShow			: INT;
                                                                       
	//Przeciąganie podajnika knotów                                   
	bWickFeederDragingStationEnableShow					:BOOL;			//	P030_Recipes.stActRecipe.stUBL.bLidFeederDragingStationEnableShow					// Aktywacja przeciagania formatek pod podajnikem płatynek
	lrWickFeederDragingStationVelocityShow				:LREAL; 		//	P030_Recipes.stActRecipe.stUBL.lrLidFeederDragingStationVelocityShow				// Prędkosć przeciągania formatek pod podajnikem płatynek [0-100 %]	
    lrWickFeederDragingStationAccelerationShow			:LREAL; 		//	P030_Recipes.stActRecipe.stUBL.lrLidFeederDragingStationAccelerationShow		// Przyspieszenie przeciągania formatek pod podajnikem płatynek 	
    lrWickFeederDragingStationDecelerationShow			:LREAL; 		//	P030_Recipes.stActRecipe.stUBL.lrLidFeederDragingStationDecelerationShow		// Zmniejszenie prędkości przeciągania formatek pod podajnikem płatynek 	
                                                                      
	//Podajnik platynek                                                 //
	bLidFeederEnableShow								:BOOL;			//	P030_Recipes.stActRecipe.stUBL.bLidFeederEnableShow				// Zezwolenie na pracę podajnika platynek 
	bLidFeederHeaterEnableShow							:BOOL;			//	P030_Recipes.stActRecipe.stUBL.bLidFeederHeaterEnableShow			// Zezwolenie na prace grzałki podajnika platynek 
	lrLidFeederHeightPosSVShow							:LREAL;			//	P030_Recipes.stActRecipe.stUBL.lrLidFeederHeightPosSVShow			// Wysokość na której ma znajdować się podajnik platynek
	iLidFeederHeatingTimeShow							:INT; 			//	P030_Recipes.stActRecipe.stUBL.iLidFeederHeatingTimeShow			// Czas zgrzewania wstępnego podajnika platynek [ms]
	iLidFeederTempHisteresisShow						:INT;			//	P030_Recipes.stActRecipe.stUBL.iLidFeederTempHisteresisShow		// Histereza poprawnej temperatury grzałki podajnika platynek 1 (+/- *C), po jej przekroczeniu grzałka wpada w błąd
	iLidFeeder1TempSVShow								:INT;			//	P030_Recipes.stActRecipe.stUBL.iLidFeeder1TempSVShow				// Temperatura zadana grzałki podajnika platynek 1
	iLidFeeder2TempSVShow								:INT;			//	P030_Recipes.stActRecipe.stUBL.iLidFeeder2TempSVShow				// Temperatura zadana grzałki podajnika platynek 2
                                                                        //
	//Przeciąganie podajnika platynek                                   //
	bLidFeederDragingStationEnableShow					: BOOL;			//	P030_Recipes.stActRecipe.stUBL.bLidFeederDragingStationEnableShow					// Aktywacja przeciagania formatek pod podajnikem płatynek
	lrLidFeederDragingStationVelocityShow				: LREAL; 		//	P030_Recipes.stActRecipe.stUBL.lrLidFeederDragingStationVelocityShow				// Prędkosć przeciągania formatek pod podajnikem płatynek [0-100 %]	
    lrLidFeederDragingStationAccelerationShow			: LREAL; 		//	P030_Recipes.stActRecipe.stUBL.lrLidFeederDragingStationAccelerationShow		// Przyspieszenie przeciągania formatek pod podajnikem płatynek 	
    lrLidFeederDragingStationDecelerationShow			: LREAL; 		//	P030_Recipes.stActRecipe.stUBL.lrLidFeederDragingStationDecelerationShow		// Zmniejszenie prędkości przeciągania formatek pod podajnikem płatynek 	

                                                                       //
	//Sprawdzanie platynek                                              //
	bLidPuttedCheckEnableShow      						: BOOL;  		//	P030_Recipes.stActRecipe.stUBL.bLidPuttedCheckEnableShow   			// Zezwolenie na prace stacji sprawdzania nakrętek
    lrLidPuttedCheckHeightSVShow 	 					: LREAL;        //    P030_Recipes.stActRecipe.stUBL.lrLidPuttedCheckHeightSVShow			
	lrLidPuttedCheckPositionShow						: LREAL;		//	P030_Recipes.stActRecipe.stUBL.lrLidPuttedCheckPositionShow			// Pozycka sprawdzania platynki
	lrLidPuttedCheckAreaShow							: LREAL;		//	P030_Recipes.stActRecipe.stUBL.lrLidPuttedCheckAreaShow				// [-50...50]  lrLidPuttedCheckPosition +- lrLidPuttedCheckArea. Granica monitorowania 
	iLidPuttedCheckProgramShow							: INT;			//	P030_Recipes.stActRecipe.stUBL.iLidPuttedCheckProgramShow				// Program czujnika wizyjnego 0-20
                                                                        //
	//Zgrzewanie                                                        //
	bLidSealerEnableShow								: BOOL;			//	P030_Recipes.stActRecipe.stUBL.bLidSealerEnableShow				// Zezwolenie na pracę podajnika 
    bLidSealerHeaterEnableShow							: BOOL;			//	P030_Recipes.stActRecipe.stUBL.bLidSealerHeaterEnableShow			// Zezwolenie na prace grzałki  
    iLidSealerHeatingTimeShow							: INT;			//	P030_Recipes.stActRecipe.stUBL.iLidSealerHeatingTimeShow			// Czas zgrzewania  [ms]
	lrLidSealerPressureShow								: LREAL;		//	P030_Recipes.stActRecipe.stUBL.lrLidSealerPressureShow				//	Siła zgrzewania [kg] 
  	lrLidSealerHeightPosSVShow							: LREAL;		//	P030_Recipes.stActRecipe.stUBL.lrLidSealerHeightPosSVShow			// Wysokoć na której ma znajdować się grzałka
	iLidSealerTempHisteresisShow						: INT;			//	P030_Recipes.stActRecipe.stUBL.iLidSealerTempHisteresisShow		// Histereza poprawnej temperatury grzałki (+/- *C), po jej przekroczeniu grzałka wpada w błšd
   	iLidSealer1TempSVShow								: INT;			//	P030_Recipes.stActRecipe.stUBL.iLidSealer1TempSVShow				// Temperatura zadana grzałki 1                                                               
  	iLidSealer2TempSVShow								: INT;			//	P030_Recipes.stActRecipe.stUBL.iLidSealer2TempSVShow				// Temperatura zadana grzałki 2
                                                                        //
	//Przeciąganie zgrzewania                                           //
	bLidSealerDragingStationEnableShow					: BOOL;			//	P030_Recipes.stActRecipe.stUBL.bLidSealerDragingStationEnableShow					// Aktywacja przeciagania formatek pod zakrecarkami
	lrLidSealerDragingStationVelocityShow				: LREAL; 		//	P030_Recipes.stActRecipe.stUBL.lrLidSealerDragingStationVelocityShow				// Prędkosć przeciągania formatek pod zakręcarkami [0-100 %]
    lrLidSealerDragingStationAccelerationShow			: LREAL; 		//	P030_Recipes.stActRecipe.stUBL.lrLidSealerDragingStationAccelerationShow		// Przyspieszenie przeciągania formatek pod podajnikem płatynek 	
    lrLidSealerDragingStationDecelerationShow			: LREAL; 		//	P030_Recipes.stActRecipe.stUBL.lrLidSealerDragingStationDecelerationShow		// Zmniejszenie prędkości przeciągania formatek pod podajnikem płatynek 	
                                                                        //
	//Szlaban podawania zamknięć                            			//	
	bCapFeederGateEnableShow							:BOOL;			//	P030_Recipes.stActRecipe.stUBL.bCapFeederGateEnableShow				// Aktywacja 
	iCapFeederGateBlockingTimeShow						:INT;			//	P030_Recipes.stActRecipe.stUBL.iCapFeederGateBlockingTimeShow		// Czas blokowania
                                                                        //
	//[H] Podajnik zamknięć                        				        //
	bCapFeederEnableShow								:BOOL;			//	P030_Recipes.stActRecipe.stUBL.bCapFeederEnableShow							// [H] Aktywacja
    lrCapFeederHeightPosSVShow							:LREAL:=140;	//	P030_Recipes.stActRecipe.stUBL.lrCapFeederHeightPosSVShow						// [H] Pozycja
	iCapFeederTimeDelayOnShow							:INT; 			//	P030_Recipes.stActRecipe.stUBL.iCapFeederTimeDelayOnShow						// [H] Opóźnienie włączenia
	iCapFeederTimeDelayOffShow							:INT; 			//	P030_Recipes.stActRecipe.stUBL.iCapFeederTimeDelayOffShow						// [H] Opóźnienie wyłączenia
	iCapFeederTimeToEmptySleeveErrorShow				:INT;			//	P030_Recipes.stActRecipe.stUBL.iCapFeederTimeToEmptySleeveErrorShow			// [H] Czas do alarmu pustego rękawa [s] (10-120 s)
                                                                        //
	//Sorter nasadek                                                    //
	//Zmienne z innego sterownika                                       //
	bCapSorterOnlyWeightOKEnableShow					:BOOL;			//	P030_Recipes.stActRecipe.stUBL.bCapSorterOnlyWeightOKEnableShow		// Nakładanie zamknięć tylko na opakowania z waga OK
	                                                                    //
	//Przeciąganie pod sorterem nasadek                                 //
	bCapSorterDragEnableShow							:BOOL;			//	P030_Recipes.stActRecipe.stUBL.bCapSorterDragEnableShow				// [H] Aktywacja
	lrCapSorterDragVelocityShow							:LREAL; 		//	P030_Recipes.stActRecipe.stUBL.lrCapSorterDragVelocityShow				// Prędkość
 	lrCapSorterDragAccelerationShow						:LREAL;			//	P030_Recipes.stActRecipe.stUBL.lrCapSorterDragAccelerationShow			// Przyspieszenie 
	lrCapSorterDragDecelerationShow						:LREAL;			//	P030_Recipes.stActRecipe.stUBL.lrCapSorterDragDecelerationShow			// Hamowanie
                                 				                        //
	//Sprawdzanie nasadki                                      			//	
	bCapPuttedCheckEnableShow							:BOOL;			//	P030_Recipes.stActRecipe.stUBL.bCapPuttedCheckEnableShow				// Aktywacja
    lrCapPuttedCheckHeightPosSVShow						:LREAL:=69;		//	P030_Recipes.stActRecipe.stUBL.lrCapPuttedCheckHeightPosSVShow			// Pozycja
                                 					                    //
	//Zakrecarka szczekowa (Zachować kolejność i opisy!)                //
	bGripperScrewer1EnableShow							:BOOL;			//	P030_Recipes.stActRecipe.stUBL.bGripperScrewer1EnableShow								// Aktywacja 1
	lrGripperScrewingTightTorqueShow					:LREAL;  		//	P030_Recipes.stActRecipe.stUBL.lrGripperScrewingTightTorqueShow						// Nastawa momentu zakręcania [Nm]
	bGripperScrewer2EnableShow							:BOOL;			//	P030_Recipes.stActRecipe.stUBL.bGripperScrewer2EnableShow								// Aktywacja 2
	lrGripperScrewing2TightTorqueShow					:LREAL;  		//	P030_Recipes.stActRecipe.stUBL.lrGripperScrewing2TightTorqueShow						// Nastawa momentu zakręcania 2 [Nm]
	iGripperScrewer1ToolShow							:INT;			//	P030_Recipes.stActRecipe.stUBL.iGripperScrewer1ToolShow								// Wybór narzędzia (1-5), opisy w tablicy AsGripperScrewerTool	
 	lrGripperScrewer1VelocityShow						:LREAL:=6000; 	//	P030_Recipes.stActRecipe.stUBL.lrGripperScrewer1VelocityShow							// Prędkość zakręcania [rpm]
	nGripperScrewer1TightTimeShow						:INT:=100;  	//	P030_Recipes.stActRecipe.stUBL.nGripperScrewer1TightTimeShow							// Czas przytrzymania podczas dokręcania [ms] 	
	iGripperScrewer1StartDelayShow						:INT;			//	P030_Recipes.stActRecipe.stUBL.iGripperScrewer1StartDelayShow							// Zwoka przed zakręcaniem			
	lrGripperScrewerReadyPositionShow					:LREAL := 250;  //	P030_Recipes.stActRecipe.stUBL.lrGripperScrewerReadyPositionShow						// Pozycja gotowości
	lrGripperScrewerPushingCapPositionShow				:LREAL := 250;  //	P030_Recipes.stActRecipe.stUBL.lrGripperScrewerPushingCapPositionShow					// Pozycja docisku  
    lrGripperScrewerScrewingCapPositionShow				:LREAL := 250;  //	P030_Recipes.stActRecipe.stUBL.lrGripperScrewerScrewingCapPositionShow					// Pozycja zakręcania	
    lrGripperScrewerFindScrewPositionShow				:LREAL := 250;  //	P030_Recipes.stActRecipe.stUBL.lrGripperScrewerScrewingCapPositionShow					// Pozycja zakręcania	
	lrGripperScrewerPressureShow						:LREAL;			//	P030_Recipes.stActRecipe.stUBL.lrGripperScrewerPressureShow							// Siła chwytaka nasadki (0.0 kg)
	lrGripperScrewerCatchPressureShow 					:LREAL;			//	P030_Recipes.stActRecipe.stUBL.lrGripperScrewerCatchPressureShow 						// Siła chwytaka butelki (0.0 kg)
	lrDispencerCatchPressureShow 						:LREAL;			//	P030_Recipes.stActRecipe.stUBL.lrDispencerCatchPressureShow 							// Siła chwytaka butelki pod dozownikami (0.0 kg)
	lrGripperScrewerPressureExhaustLevelShow			:LREAL;			//	P030_Recipes.stActRecipe.stUBL.lrGripperScrewerPressureExhaustLevelShow				// Prędkość zamykania chwytaka nasadki (0.0-100.0 %)
	lrGripperScrewerCatchPressureExhaustLevelShow		:LREAL;			//	P030_Recipes.stActRecipe.stUBL.lrGripperScrewerCatchPressureExhaustLevelShow			// Prędkość zamykania chwytaka opakowania (0.0-100.0 %)
	lrGripperScrewerTurnoversToFullScrewedShow			:LREAL;			//	P030_Recipes.stActRecipe.stUBL.lrGripperScrewerTurnoversToFullScrewedShow				// Opakowanie | Ilość obrotów zamknięcia [obr.] (0.5-10.0 obr.)
   	lrGripperScrewerThreadPitchShow						:LREAL;			//	P030_Recipes.stActRecipe.stUBL.lrGripperScrewerThreadPitchShow							// Opakowanie | Skok gwintu [mm] (0.1-10.0 mm)
	lrGripperScrewerThreadTimesShow						:LREAL;			//	P030_Recipes.stActRecipe.stUBL.lrGripperScrewerThreadTimesShow							// Opakowanie | Krotność gwintu [x] (1-10 x)                       		
	nGripperScrewerCatchHeightSVShow					:LREAL:=86;  		//	P030_Recipes.stActRecipe.stUBL.nGripperScrewerCatchHeightSVShow						// Pozycja chwytaka opakowań
	bGripperScrewer1FindScrewShow						:BOOL; 			//	P030_Recipes.stActRecipe.stUBL.bGripperScrewer1FindScrewShow							// Szukanie gwintu w pozycji zakręcania	
	bGripperScrewer1Option4Show							:BOOL;			//	P030_Recipes.stActRecipe.stUBL.bGripperScrewer1Option4Show								// Szukanie gwintu w pozycji dociskania	
	lrGripperScrewer1FindingScrewDegreeShow				:LREAL; 		//	P030_Recipes.stActRecipe.stUBL.lrGripperScrewer1FindingScrewDegreeShow					// Kąt szukania gwintu (max. dla opcji szukania gwintu z czuj. wys.)	
	bGripperScrewer1Option1Show							:BOOL;			//	P030_Recipes.stActRecipe.stUBL.bGripperScrewer1Option1Show								// Otwarty chwytak przy szukaniu gwintu	
	bGripperScrewer1Option2Show							:BOOL;			//	P030_Recipes.stActRecipe.stUBL.bGripperScrewer1Option2Show								// Obrót do tyłu w pozycji dociskania (w trakcie przejazdu do poz. doc.)
	bGripperScrewer1Option3Show							:BOOL;			//	P030_Recipes.stActRecipe.stUBL.bGripperScrewer1Option3Show								// Dodatkowy ruch chwytakiem przed zakręceniem  (w poz. doc.)	
	bGripperScrewer1Option5Show							:BOOL;			//	P030_Recipes.stActRecipe.stUBL.bGripperScrewer1Option5Show								// Szukanie gwintu z czujnikiem wysokości
	bGripperScrewer1Option6Show							:BOOL;			//	P030_Recipes.stActRecipe.stUBL.bGripperScrewer1Option6Show								// Obrót z pozycji docisku do zakręcania
 	bGripperScrewer1Option7Show							:BOOL;			//	P030_Recipes.stActRecipe.stUBL.bGripperScrewer1Option7Show								// Tryb momentowy	
	                                                                    //
	//Przeciaganie formatek pod zakrecarkami                            //
	bBottleDragingStationEnableShow						:BOOL;			//	P030_Recipes.stActRecipe.stUBL.bBottleDragingStationEnableShow				// [H] Aktywacja 
	lrBottleDragingStationVelocityShow					:LREAL; 		//	P030_Recipes.stActRecipe.stUBL.lrBottleDragingStationVelocityShow		// Prędkość
	                                                                    //
	//Sprawdzanie zakręcania                                            //
	bCapCorrectCheckEnableShow							:BOOL;			//	P030_Recipes.stActRecipe.stUBL.bCapCorrectCheckEnableShow					// Aktywacja
    lrCapCorrectCheckHeightPosSVShow					:LREAL:=69;		//	P030_Recipes.stActRecipe.stUBL.lrCapCorrectCheckHeightPosSVShow			// Pozycja
	bCapCorrectCheckCameraEnableShow      				:BOOL;  		//	P030_Recipes.stActRecipe.stUBL.bCapCorrectCheckCameraEnableShow 		// Aktywacja sprawdzania orientacji nasadki
	iCapCorrectCheckCameraProgramShow					:INT;			//	P030_Recipes.stActRecipe.stUBL.iCapCorrectCheckCameraProgramShow		// Program czujnika wizyjnego 0-20
	                                                                    //
	                                                                    //
	//Robot butelek                                                     //
	bBottleTransferEnableShow							:BOOL; 			//	P030_Recipes.stActRecipe.stUBL.bBottleTransferEnableShow					// Aktywacja
	nBottleTransferProgramShow							:UINT; 			//	P030_Recipes.stActRecipe.stUBL.nBottleTransferProgramShow					// [H] Program robota	
	iBottleTransferPickOffsetXShow 						:INT;			//	P030_Recipes.stActRecipe.stUBL.iBottleTransferPickOffsetXShow 				// Offset X pozycji pobrania
	iBottleTransferPickOffsetYShow 						:INT;			//	P030_Recipes.stActRecipe.stUBL.iBottleTransferPickOffsetYShow 				// Offset Y pozycji pobrania  
	iBottleTransferPickOffsetZShow 						:INT; 			//	P030_Recipes.stActRecipe.stUBL.iBottleTransferPickOffsetZShow 				// Offset Z pozycji pobrania
	iBottleTransferPick2OffsetXShow						:INT;			//	P030_Recipes.stActRecipe.stUBL.iBottleTransferPick2OffsetXShow				// Offset X 2 pozycji pobrania
	iBottleTransferPick2OffsetYShow						:INT;  			//	P030_Recipes.stActRecipe.stUBL.iBottleTransferPick2OffsetYShow				// Offset Y 2 pozycji pobrania
	iBottleTransferPick2OffsetZShow						:INT;   		//	P030_Recipes.stActRecipe.stUBL.iBottleTransferPick2OffsetZShow				// Offset Z 2 pozycji pobrania
	iBottleTransferPlace1OffsetXShow 					:INT;			//	P030_Recipes.stActRecipe.stUBL.iBottleTransferPlace1OffsetXShow 			// Offset X pozycji etykieciarki
	iBottleTransferPlace1OffsetYShow 					:INT;  			//	P030_Recipes.stActRecipe.stUBL.iBottleTransferPlace1OffsetYShow 			// Offset Y pozycji etykieciarki
	iBottleTransferPlace1OffsetZShow 					:INT;			//	P030_Recipes.stActRecipe.stUBL.iBottleTransferPlace1OffsetZShow 			// Offset Z pozycji etykieciarki
	iBottleTransferPlace2OffsetXShow 					:INT;			//	P030_Recipes.stActRecipe.stUBL.iBottleTransferPlace2OffsetXShow 			// Offset X pozycji odrzutu
	iBottleTransferPlace2OffsetYShow					:INT;			//	P030_Recipes.stActRecipe.stUBL.iBottleTransferPlace2OffsetYShow			// Offset Y pozycji odrzutu
	iBottleTransferPlace2OffsetZShow 					:INT; 			//	P030_Recipes.stActRecipe.stUBL.iBottleTransferPlace2OffsetZShow 			// Offset Z pozycji odrzutu
	iBottleTransferSpeedShow							:INT := 10;		//	P030_Recipes.stActRecipe.stUBL.iBottleTransferSpeedShow					// Prędkość robota 	
	bBottleTransferInkJetEnableShow						:BOOL;			//	P030_Recipes.stActRecipe.stUBL.bBottleTransferInkJetEnableShow				// Przesuwanie opakowania nad drukarką (Inkjet)
  	bBottleTransferPickOnlyOneShow						:BOOL;			//	P030_Recipes.stActRecipe.stUBL.bBottleTransferPickOnlyOneShow				// [H] Pobieranie tylko 1 opakowania
 	bBottleTransferWeightEnableShow						:BOOL;			//	P030_Recipes.stActRecipe.stUBL.bBottleTransferWeightEnableShow				// Przesuwanie opakowania na wagę 
  	iBottleTransferWeightIntervalShow					:INT;			//	P030_Recipes.stActRecipe.stUBL.iBottleTransferWeightIntervalShow			// Interwał przesuwania na wagę
 	bBottleTransferRotateEnableShow						:BOOL;			//	P030_Recipes.stActRecipe.stUBL.bBottleTransferRotateEnableShow				// Obrót orientacji nasadki   

	//Przeciąganie 
	bBottleTransferAfterDragEnableShow					:BOOL;			// Aktywacja
	                                                                    //
	//Transporter odrzutu                      	                        //
	bBadBottleConveyorEnableShow						:BOOL;			//	P030_Recipes.stActRecipe.stUBL.bBadBottleConveyorEnableShow			// [H] Aktywacja
	nBadBottleConveyorVelocitySVShow					:UINT;			//	P030_Recipes.stActRecipe.stUBL.nBadBottleConveyorVelocitySVShow		// Prędkość
	                                                                    //
	//Etykieciarka                                                      //
	bLabelMachineEnableShow								:BOOL;			//	P030_Recipes.stActRecipe.stUBL.bLabelMachineEnableShow		// Aktywacja
	                                                                    //
	//Stół odbierający                                                  //
	bExitTurnTable1EnableShow							:BOOL;			//	P030_Recipes.stActRecipe.stUBL.bExitTurnTable1EnableShow		// Aktywacja
	//Transporter odbierający                                           //
	bExitConveyorEnableShow								:BOOL;			//	P030_Recipes.stActRecipe.stUBL.bExitConveyorEnableShow				// Aktywacja
	nExitConveyorVelocitySVShow							:UINT;			//	P030_Recipes.stActRecipe.stUBL.nExitConveyorVelocitySVShow			// Prędkość
	                                                                    //
	                                                                    //
	//Transportery główne                                               //
	bFormTransportersEnableShow							:BOOL;			//	P030_Recipes.stActRecipe.stUBL.bFormTransportersEnableShow							// [H] Aktywacja
	nFormTransportersDispencerVelocitySVShow			:UDINT;			//	P030_Recipes.stActRecipe.stUBL.nFormTransportersDispencerVelocitySVShow			// Prędkość transportera przed dozownikami
	nFormTransportersScrewerVelocitySVShow				:UDINT;			//	P030_Recipes.stActRecipe.stUBL.nFormTransportersScrewerVelocitySVShow				// Prędkość transportera za dozownikami
	nFormTransportersAfterCapSorterVelocitySVShow		:UDINT;			//	P030_Recipes.stActRecipe.stUBL.nFormTransportersBeforeScrewerVelocitySVShow		// Prędkość transportera przed zakręcarką
	nFormTransportersBeforeScrewerVelocitySVShow		:UDINT;			//	P030_Recipes.stActRecipe.stUBL.nFormTransportersBeforeScrewerVelocitySVShow		// Prędkość transportera przed zakręcarką
	nFormTransportersSlowerVelocitySVShow				:UDINT;			//	P030_Recipes.stActRecipe.stUBL.nFormTransportersSlowerVelocitySVShow				// Prędkość spowalniacza 
	nFormTransportersAfterScrewerVelocitySVShow			:UDINT;			//	P030_Recipes.stActRecipe.stUBL.nFormTransportersAfterScrewerVelocitySVShow			// Prędkość transportera przed zakręcarką
	nFormTransportersROPPVelocitySVShow					:UDINT;	        //    P030_Recipes.stActRecipe.stUBL.nFormTransportersROPPVelocitySVShow			
	                                                                    //
	//[H] InkJet obwodowy                                               //
	bCircularInkjetEnableShow							:BOOL;			//	P030_Recipes.stActRecipe.stUBL.bCircularInkjetEnableShow			// [H] Aktywacja
	iCircularInkjetSpeedShow							:INT;			//	P030_Recipes.stActRecipe.stUBL.iCircularInkjetSpeedShow			// [H] Prędkość 
	iCircularInkjetDelayShow							:INT;			//	P030_Recipes.stActRecipe.stUBL.iCircularInkjetDelayShow			// [H] Opóźnienie docisku rolek
	iCircularInkjetHoldShow								:INT;			//	P030_Recipes.stActRecipe.stUBL.iCircularInkjetHoldShow				// [H] Czas przytrzymania [ms]
	
	udiCounterExecuteTimeTemp: UDINT;

	//Czujniki Wenglor
	lrMinDistanceToCappedCorrectlyBottleShow			:LREAL; 
	lrMaxDistanceToCappedCorrectlyBottleShow			:LREAL;
	lrSettleTimeMeasuringCappedBottleShow 				:UINT;
	bWenglorSensorCapPuttedShow							:BOOL:=FALSE;
	bWenglorSensorCapCorrectShow						:BOOL:=FALSE;
	bWenglorSensorCapModeShow							:UINT;
	
	//	(***MAIN***)
	//AnRFIDCardNumberShow							:ARRAY [1..100] OF ULINT;	// [H] Tabela numerów formatek 
	//AnRFIDWeightShow								:ARRAY [1..100] OF LREAL;	// [H] Tabela wag formatek	
	
	
END_VAR

VAR_GLOBAL PERSISTENT
	
	(***MAIN***)
	AnRFIDCardNumberShow							:ARRAY [1..100] OF ULINT;	// [H] Tabela numerów formatek 
	AnRFIDWeightShow								:ARRAY [1..100] OF LREAL;	// [H] Tabela wag formatek		

    
	udiCounterGlobal								:UDINT; 					// Globalny licznik [szt.]
	udiCounterGlobalBadBottles						:UDINT;						// Globalny licznik odrzutu [szt.]

	(*****P02_Dispencers****)		
	lrFormsDragingLeftStartPosition					:LREAL;
	lrFormsDragingLeftEndPosition					:LREAL;
	lrFormsDragingRightStartPosition				:LREAL;
	lrFormsDragingRightEndPosition					:LREAL;

	(*****P10_GripperScrewer****)		
	lrBottleDragingStationStartPosition				:LREAL;
	lrBottleDragingStationEndPosition				:LREAL;	
	udiGripperScrewerToolCounter					:UDINT; 	// Licznik kasowalny dla 

	(*****P07_ROPP****)		
	lrROPPDragStationStartPosition					:LREAL;
	lrROPPDragStationEndPosition					:LREAL;	
	
	(*****P08_CapSorter****)		
	lrCapSorterDragStationStartPosition				:LREAL;
	lrCapSorterDragStationEndPosition				:LREAL;	
		
		
	(*****P10_LidSealer****)		
	lrFeedingDragingStationStartPosition				:LREAL;
	lrFeedingDragingStationEndPosition					:LREAL;	
	lrSealingDragingStationStartPosition				:LREAL;
	lrSealingDragingStationEndPosition					:LREAL;		
	
	lrWickFeedingDragingStationStartPosition				:LREAL;
	lrWickFeedingDragingStationEndPosition					:LREAL;	
	
END_VAR

// ---- GVLs/VIS_CP.TcGVL

VAR_GLOBAL
	
	(*****P07_CapPusher********)	  
	IbCapPusher0DoorsOpen 				AT %I* :BOOL;
	//Szlaban
	bCapPusherManualGate						:BOOL;						// Szlaban formatki		
	
	//Podajnik 
	iCapPusherFeederState						:INT;						// Stan
	sCapPusherFeederState						:STRING;					// Stan
    bCapPusherFeederHoming						:BOOL;						// Bazowanie
 	bCapPusherFeederRun							:BOOL; 						// Cykl
	bCapPusherFeederIgnoreErrors				:BOOL;					 	// Ignoruj błędy
	bCapPusherFeederHeightSet					:BOOL;						// Ustaw
	bCapPusherFeederManualSorterEngine			:BOOL;						// Silnik
	bCapPusherFeederManualSorterVibrator		:BOOL;						// Wibrator
	bCapPusherFeederManualSorterVibrator2		:BOOL;						// Wibrator
	bCapPusherFeederManualSorterAir				:BOOL;						// Wydmuch

	//Zakrecanie
	iCapPusherState								:INT;						// Stan
	sCapPusherState								:STRING;					// Stan
    bCapPusherHoming							:BOOL;						// Bazowanie
 	bCapPusherRun								:BOOL; 						// Cykl
	bCapPusherIgnoreErrors						:BOOL;					 	// Ignoruj błędy
	bCapPusherHeightSet							:BOOL;						// Ustaw
	bCapPusherManualPusher						:BOOL;						// Wbijak
	bCapPusherManualBlockActuator				:BOOL;						// Boczny	
	bCapPusherManualFormPositioning				:BOOL;						// Pozycjonowanie formatek
	
	(*****P00_Recipes*******)	  
	//Szlaban

	//Podajnik                     				
	iCapPusherFeederTimeDelayOnShow				:INT; 						// Opóźnienie włączenia
	iCapPusherFeederTimeDelayOffShow			:INT; 						// Opóźnienie wyłączenia
	iCapPusherFeederTimeToEmptySleeveErrorShow	:INT;						// Czas do alarmu pustego rękawa [s] (10-120 s)

	//Zakrecanie                    				
	bCapPusherEnableShow						:BOOL;						// Aktywacja
	iCapPusherTimeShow							:INT; 						// Czas wibjania
	iCapPusherTime2Show							:INT;						// Czas 2

END_VAR

// ---- GVLs/VIS_M.TcGVL
{attribute 'qualified_only'}
VAR_GLOBAL
	

	iPuckHeight	:INT:=85; 			// Wysokość wkładki w formatce razem z formatką (0-100mm)    // Uzywane do pozycji minimalnych stacji   


END_VAR

// ---- GVLs/VIS_RFID.TcGVL

VAR_GLOBAL
	sRFIDInfo											:	STRING;	// Opis sumy błędów RFID
	bRFIDCheckReset										:	BOOL;	// Reset liczników
	
	iRFIDCheckNumberOfFormsAfterWeighting				:	INT; //Liczba formatek po przeważaniu
	iRFIDCheckNumberOfFormsExecute						:	INT; //Liczba formatek na lini w czasie cyklu
	
	AStRFIDCheck										:	ARRAY [1..100] OF S_RFIDCheck;		
															(*	iNumber				: INT;		//Numer RFID	
																iReaded1			: INT;		//Odczytano z czytnika nr 1 (przed dozownikami) 
																iReaded2			: INT;		//Odczytano z czytnika nr 2	(przed wagami)
																iReaded3			: INT;		//Odczytano z czytnika nr 3	(przed zakrecarka)
																iReaded4			: INT;		//Odczytano z czytnika nr 4 (za zakrecarka)
																iReaded5			: INT;		//Odczytano z czytnika nr 5	(robot)*)
																
	iRFIDCheckDispencerWarning							:	INT;	// Liczba błędnych rejestrów dozowniki
	iRFIDCheckWeightWarning								:	INT;	// Liczba błędnych rejestrów wagi
	iRFIDCheckBeforeScrewerWarning						:	INT;	// Liczba błędnych rejestrów zakrecarki
	iRFIDCheckAfterScrewerWarning						:	INT;	// Liczba błędnych rejestrów test zakrecania
	iRFIDCheckBottleTransferWarning						:	INT;	// Liczba błędnych rejestrów robot
								
END_VAR

// ---- GVLs/VIS_ROPP.TcGVL

VAR_GLOBAL
	
	(*****P07_ROPP********)	  

	//Spowalniacz
	iROPPSlowerState							:INT;						// Stan pracy 
	sROPPSlowerState							:STRING;					// Stan pracy 
	nROPPSlowerVelocityCV						:INT;						// Aktualna predkość
	bROPPSlowerManualCmdStart					:BOOL; 						// Spowalniacz

	//Podajnik 
	iROPPFeederState							:INT;						// Stan
	sROPPFeederState							:STRING;					// Stan
    bROPPFeederHoming							:BOOL;						// Bazowanie
 	bROPPFeederRun								:BOOL; 						// Cykl
	bROPPFeederIgnoreErrors						:BOOL;					 	// Ignoruj błędy
	bROPPFeederHeightSet						:BOOL;						// Ustaw
	bROPPFeederManualHeightUp					:BOOL;						// Do góry
	bROPPFeederManualHeightDown					:BOOL;						// Na doł
	bROPPFeederManualSorterEngine				:BOOL;						// Silnik
	bROPPFeederManualSorterVibrator				:BOOL;						// Wibrator
	bROPPFeederManualSorterAir					:BOOL;						// Wydmuch
	bROPPFeederManualSorterAir2					:BOOL;						// Wydmuch 2
	bROPPFeederManualConveyorStart				:BOOL;						// Zasyp start
	bROPPFeederManualConveyorStop				:BOOL;						// Zasyp stop
	lrROPPFeederHeightCV						:LREAL;						// Aktualna wyskokość 

	//Sprawdzanie kapsla
	bROPPPuttedCheckOK							:BOOL;						// Kapsel nałożony

	//Stoper
	bROPPStoperBeforeManualActuator				:BOOL;						// Stoper
	bROPPStoperAfterManualActuator				:BOOL;						// Stoper

	//Przeciąganie formatek 
	iROPPDragState								:INT;						// Stan
	sROPPDragState								:STRING;					// Stan
	bROPPDragRun								:BOOL;						// Cykl
	bROPPDragHoming								:BOOL;						// Bazowanie 
	bROPPDragIgnoreError						:BOOL;						// Ignoruj błędy
	bROPPDragManualFork							:BOOL;						// Podnosnik
	bROPPDragManualLead							:BOOL;						// Prowadzenie
	bROPPDragManualLeft							:BOOL;						// Do przodu
	bROPPDragManualRight						:BOOL;						// Do tyłu
	lrROPPDragPositionCV						:LREAL;						// Aktualna pozycja

	//Zakrecanie
	iROPPCappingState							:INT;						// Stan
	sROPPCappingState							:STRING;					// Stan
    bROPPCappingHoming							:BOOL;						// Bazowanie
 	bROPPCappingRun1							:BOOL; 						// Cykl 1
 	bROPPCappingRun2							:BOOL; 						// Cykl 2
	bROPPCappingIgnoreErrors					:BOOL;					 	// Ignoruj błędy
	bROPPCappingHeightSet						:BOOL;						// Ustaw
	AsROPPCappingTool							:ARRAY [1..10] OF STRING;	// Głowica (1-Opis_narzędzia_nr_1, 2-Opis_narzędzia_nr_2)
	bROPPCappingManualHeightUp					:BOOL;						// Do góry
	bROPPCappingManualHeightDown				:BOOL;						// Na doł
	bROPPCappingManualEngine1					:BOOL;						// Głowica 1 - Silnik
	bROPPCappingManualEngine2					:BOOL;						// Głowica 2 - Silnik
	bROPPCappingManualCapping1Tool1Actuator		:BOOL;						// Głowica 1 - Narzędzie 1 - Siłownik	
	bROPPCappingManualCapping2Tool1Actuator		:BOOL;						// Głowica 2 - Narzędzie 1 - Siłownik		
	bROPPCappingManualCapping12Tool1BlockActuator:BOOL;						// Głowica 1 i 2 - Narzędzie - Blokada		
	bROPPCappingManualCappingBlockActuator		:BOOL;						// Blokada podnośnika			
	bROPPCappingManualCapping1Tool2Down			:BOOL;						// Głowica 1 - Narzędzie 2 - Dół	
	bROPPCappingManualCapping1Tool2Tight		:BOOL;						// Głowica 1 - Narzędzie 2 - Zaciśnij		
	bROPPCappingManualCapping1Tool2Realese		:BOOL;						// Głowica 1 - Narzędzie 2 - Odpuść
	bROPPCappingManualCapping2Tool2Down			:BOOL;						// Głowica 2 - Narzędzie 2 - Dół
	bROPPCappingManualCapping2Tool2Tight		:BOOL;						// Głowica 2 - Narzędzie 2 - Zaciśnij	
	bROPPCappingManualCapping2Tool2Realese		:BOOL;						// Głowica 2 - Narzędzie 2 - Odpuść	
	bROPPCappingManualFormPositioning			:BOOL;						// Pozycjonowanie formatek
	lrROPPCappingHeightCV						:LREAL;						// Aktualna wysokość 

	//Sprawdzanie kapsla 
	bROPPCappingCheckOK							:BOOL;						// Kapsel OK po zakręceniu
	
	(*****P00_Recipes*******)	  
	//Spowalniacz
	bROPPSlowerEnableShow						:BOOL;						// Aktywacja
	nROPPSlowerVelocitySVShow					:UDINT;						// Prędkość 

	//Podajnik                     				
	bROPPFeederEnableShow						:BOOL;						// Aktywacja
    lrROPPFeederHeightPosSVShow					:LREAL:=140;				// Pozycja
	iROPPFeederTimeDelayOnShow					:INT; 						// Opóźnienie włączenia
	iROPPFeederTimeDelayOffShow					:INT; 						// Opóźnienie wyłączenia
	iROPPFeederTimeToEmptySleeveErrorShow		:INT;						// Czas do alarmu pustego rękawa [s] (10-120 s)

	//Przeciąganie 
	bROPPDragEnableShow							:BOOL;						// Aktywacja
	lrROPPDragVelocityShow						:LREAL; 					// Prędkość
 	lrROPPDragAccelerationShow					:LREAL;						// Przyspieszenie 
	lrROPPDragDecelerationShow					:LREAL;						// Hamowanie

	//Zakrecanie                    				
	bROPPCappingEnableShow						:BOOL;						// Aktywacja
    lrROPPCappingHeightPosSVShow				:LREAL:=140;				// Pozycja
   	lrROPPCappingVelocitySVShow					:UDINT;						// Prędkość
	iROPPCappingTimeShow						:INT; 						// Czas 1
	iROPPCappingTime2Show						:INT;						// Czas 2
	iROPPCapping1ToolShow						:INT;						// Wybór narzędzia (1-2), opisy w tablicy AsROPPCappingTool	1-Głowica zakręcająca, 2-Głowica zaciskająca

END_VAR

// ---- GVLs/VIS_RS.TcGVL
{attribute 'qualified_only'}
VAR_GLOBAL
	
	
	(*****P10_RollerScrewer********)          
	//Szlaban
	bRollerScrewerManualFormGate						: BOOL;		// Szlaban formatki		

	//Zakręcarka rolkowa      			
	iRollerScrewerState									: INT; 		
	sRollerScrewerState									: STRING;
	bRollerScrewerHoming								: BOOL; 	
	bRollerScrewerHeightSet								: BOOL; 								
    bRollerScrewerIgnoreErrors							: BOOL; 	
    bRollerScrewerRun									: BOOL; 					
	bRollerScrewerManualRight							: BOOL;  	// Obrót w lewo
    bRollerScrewerManualLeft							: BOOL;   	// Obrót w prawo
	bRollerScrewerManualPressingTopActuator				: BOOL; 	// Docisk
	bRollerScrewerManualPressingRollsActuator			: BOOL;		// Rolki
    bRollerScrewerManualHeightUp						: BOOL; 						
    bRollerScrewerManualHeightDown						: BOOL; 	
	lrRollerScrewerHeightCV								: LREAL; 	// Aktualna wysokoć 
	bRollerScrewerCapPuttedCheckOK						: BOOL;		// Czujnik wykrycia nasadki przed zakręcarką					// Plantyka OK

	//Chytak zakrecarki rolkowej                    			
	iRollerScrewerCatchState							: INT;  		
 	sRollerScrewerCatchState							: STRING;
    bRollerScrewerCatchHeightSet						: BOOL;								
    lrRollerScrewerCatchHeightCV						: LREAL;  						  	
	bRollerScrewerCatchManualActuator					: BOOL;  						
    bRollerScrewerCatchManualUp							: BOOL;  							
    bRollerScrewerCatchManualDown						: BOOL;  							

	(*Receptury*)
	//Ciśnienia - nie wiadomo czy będą
	lrRollerScrewerCatchPressureShow 					:LREAL;			//	Siła zakręcarki rolkowej
	lrRollerScrewerPressingRollsPressureShow 			:LREAL;			//	Siła docisku rolek zakręcarki rolkowej
	lrRollerScrewerPressingTopPressureShow 				:LREAL;			//	Siła docisku górnego zakręcarki rolkowej	
	//Zakręcarka rolkowa
	bRollerScrewerEnableShow							: BOOL;			// Aktywacja
	bRollerScrewerFindScrewShow							: BOOL; 		// Aktywacja szukania gwintu
	lrRollerScrewerFindingScrewDegreeShow				: LREAL; 		// Kąt szukania gwintu
	lrRollerScrewerVelocityShow							: LREAL:=50; 	// Prędkość zakręcania [rpm]
	iRollerScrewerTightTimeShow							: INT:=100;  	// Czas przytrzymania nakrętki z zadanym momentem [ms] 
	lrRollerScrewingTightTorqueShow						: LREAL;  		// Nastawa momentu zakręcania [Nm]
    lrRollerScrewerHeightPosSVShow						: LREAL:=72;	// Pozycja stacji
	uiRollerScrewerTopActuatorTimeDelayOffShow			: UINT;  		// Czas po którym odpusczany jest docisk górny
	//Chwytak zakręcarki rolkowej                               			
	lrRollerScrewerCatchHeightSVShow					: LREAL:=36; 								// Pozycja chwytka


END_VAR

// ---- POUs/FB/AxisControl/AX8000/I_AxisControlPhysical.TcIO
//==================================================================================================
//							Beckhoff Automation Poland
//									03.01.2023
//
// Code owner: TG
//
// Sample interface to handle physical axis
//
// Used libraries: 
//	Tc2_MC2								|| 3.3.48.0
//
//  v1.0	|| TC v 3.1.4024.35		|| First edition
//==================================================================================================
INTERFACE I_AxisControlPhysical

METHOD DeletePositionOffset 					: REFERENCE TO Tc2_MC2.ST_McOutputs
VAR_INPUT
	bExecute									: BOOL;
	eFeedback									: Tc2_MC2_Drive.E_PositionOffsetFeedback;
	eMemory										: Tc2_MC2_Drive.E_PositionOffsetMemory;
END_VAR
END_METHOD

METHOD DeletePositionOffsetClear 				: BOOL
END_METHOD

METHOD DeletePositionOffsetEncoder 				: REFERENCE TO Tc2_MC2.ST_McOutputs
VAR_INPUT
	bExecute									: BOOL;
END_VAR
END_METHOD

METHOD DeletePositionOffsetEx 					: BOOL
VAR_INPUT
	eFeedback									: Tc2_MC2_Drive.E_PositionOffsetFeedback;
	eMemory										: Tc2_MC2_Drive.E_PositionOffsetMemory;
END_VAR
END_METHOD

PROPERTY pDeletePosOffs 							: REFERENCE TO ST_McOutputs
GET
END_GET
SET
END_SET
END_PROPERTY

PROPERTY pDriveAddress 							: REFERENCE TO Tc2_MC2.ST_DriveAddress
GET
END_GET
END_PROPERTY

PROPERTY pDriveRef 								: REFERENCE TO Tc2_EtherCAT.ST_DriveRef
GET
END_GET
END_PROPERTY

PROPERTY pSetPosOffs 							: REFERENCE TO ST_McOutputs
GET
END_GET
SET
END_SET
END_PROPERTY

METHOD ReadI2T 							: BOOL
END_METHOD

METHOD ReadMotionPowerData 						: BOOL
END_METHOD

METHOD ReadMotorTorque 							: LREAL
END_METHOD

METHOD SetPositionOffset 						: REFERENCE TO Tc2_MC2.ST_McOutputs
VAR_INPUT
	bExecute									: BOOL;
	fPosition									: LREAL;
	bRelative									: BOOL;
	eFeedback									: Tc2_MC2_Drive.E_PositionOffsetFeedback;
	eMemory										: Tc2_MC2_Drive.E_PositionOffsetMemory;
END_VAR
END_METHOD

METHOD SetPositionOffsetClear 					: BOOL
END_METHOD

METHOD SetPositionOffsetEncoderAbs 				: REFERENCE TO Tc2_MC2.ST_McOutputs
VAR_INPUT
	bExecute									: BOOL;
	fPosition									: LREAL;
END_VAR
END_METHOD

METHOD SetPositionOffsetEncoderAbsZero 			: REFERENCE TO Tc2_MC2.ST_McOutputs
VAR_INPUT
	bExecute									: BOOL;
END_VAR
END_METHOD

METHOD SetPositionOffsetEncoderRel 				: REFERENCE TO Tc2_MC2.ST_McOutputs
VAR_INPUT
	bExecute									: BOOL;
	fPosition									: LREAL;
END_VAR
END_METHOD

METHOD SetPositionOffsetEx 						: BOOL
VAR_INPUT
	fPosition									: LREAL;
	bRelative									: BOOL;
	eFeedback									: Tc2_MC2_Drive.E_PositionOffsetFeedback;
	eMemory										: Tc2_MC2_Drive.E_PositionOffsetMemory;
END_VAR
END_METHOD

METHOD TorqueControl 							: REFERENCE TO Tc2_MC2.ST_McOutputs
VAR_INPUT
	bExecute									: BOOL;
END_VAR
END_METHOD

METHOD TorqueControlClear 						: BOOL
END_METHOD

METHOD TorqueControlEx 							: BOOL
END_METHOD

END_INTERFACE

// ---- POUs/FB/AxisControl/Base/I_AxisControlBase.TcIO
//==================================================================================================
//							Beckhoff Automation Poland
//									03.01.2023
//
// Code owner: TG
//
// Sample Interface to handle NC Axis
//
// Used libraries: 
//	Tc2_MC2								|| 3.3.48.0
//
//  v1.0	|| TC v 3.1.4024.35		|| First edition
//==================================================================================================
INTERFACE I_AxisControlBase

PROPERTY bConsequentialError 					: BOOL
GET
END_GET
END_PROPERTY

PROPERTY bDisabled 								: BOOL
GET
END_GET
END_PROPERTY

PROPERTY bDriveError 							: BOOL
GET
END_GET
END_PROPERTY

PROPERTY bEnabled 								: BOOL
GET
END_GET
END_PROPERTY

PROPERTY bEnableNegative 						: BOOL
GET
END_GET
SET
END_SET
END_PROPERTY

PROPERTY bEnablePositive 						: BOOL
GET
END_GET
SET
END_SET
END_PROPERTY

PROPERTY bError 									: BOOL
GET
END_GET
END_PROPERTY

PROPERTY bExecuteEstop 							: BOOL
GET
END_GET
SET
END_SET
END_PROPERTY

PROPERTY bLimitSwitchStateMax 					: BOOL
GET
END_GET
SET
END_SET
END_PROPERTY

PROPERTY bLimitSwitchStateMin 					: BOOL
GET
END_GET
SET
END_SET
END_PROPERTY

PROPERTY bMoving 								: BOOL
GET
END_GET
END_PROPERTY

PROPERTY bNotMoving 								: BOOL
GET
END_GET
END_PROPERTY

PROPERTY bSimulationAxis 						: BOOL
GET
END_GET
END_PROPERTY

METHOD Disable 									: BOOL
END_METHOD

PROPERTY eBufferMode 							: MC_BufferMode
GET
END_GET
SET
END_SET
END_PROPERTY

PROPERTY eDirection 								: Tc2_MC2.MC_Direction
GET
END_GET
SET
END_SET
END_PROPERTY

PROPERTY eJogMode 								: Tc2_MC2.E_JogMode
GET
END_GET
SET
END_SET
END_PROPERTY

METHOD Enable 									: BOOL
END_METHOD

METHOD EStop 									: REFERENCE TO Tc2_MC2.ST_McOutputs
VAR_INPUT
	bExecute									: BOOL;
END_VAR
END_METHOD

METHOD EStopClear 								: BOOL
END_METHOD

METHOD EStopEx 									: BOOL
END_METHOD

PROPERTY fAcceleration 							: LREAL
GET
END_GET
SET
END_SET
END_PROPERTY

PROPERTY fActAcc 								: LREAL
GET
END_GET
END_PROPERTY

PROPERTY fActPos 								: LREAL
GET
END_GET
END_PROPERTY

PROPERTY fActTorque 								: LREAL
GET
END_GET
END_PROPERTY

PROPERTY fActVelo 								: LREAL
GET
END_GET
END_PROPERTY

PROPERTY fDeceleration 							: LREAL
GET
END_GET
SET
END_SET
END_PROPERTY

PROPERTY fDecelerationEstop 						: LREAL
GET
END_GET
SET
END_SET
END_PROPERTY

PROPERTY fDistance 								: LREAL
GET
END_GET
SET
END_SET
END_PROPERTY

PROPERTY fGearRatio 								: LREAL
GET
END_GET
SET
END_SET
END_PROPERTY

PROPERTY fJerk 									: LREAL
GET
END_GET
SET
END_SET
END_PROPERTY

PROPERTY fJerkEstop 								: LREAL
GET
END_GET
SET
END_SET
END_PROPERTY

PROPERTY fLimitSwitchPositionMax 				: LREAL
GET
END_GET
SET
END_SET
END_PROPERTY

PROPERTY fLimitSwitchPositionMin 				: LREAL
GET
END_GET
SET
END_SET
END_PROPERTY

PROPERTY fOverride 								: LREAL
GET
END_GET
SET
END_SET
END_PROPERTY

PROPERTY fPosition 								: LREAL
GET
END_GET
SET
END_SET
END_PROPERTY

PROPERTY fSetAcc 								: LREAL
GET
END_GET
END_PROPERTY

PROPERTY fSetPos 								: LREAL
GET
END_GET
END_PROPERTY

PROPERTY fSetVelo 								: LREAL
GET
END_GET
END_PROPERTY

PROPERTY fVelocity 								: LREAL
GET
END_GET
SET
END_SET
END_PROPERTY

METHOD Halt 									: REFERENCE TO Tc2_MC2.ST_McOutputs
VAR_INPUT
	bExecute									: BOOL;
END_VAR
END_METHOD

METHOD HaltClear 								: BOOL
END_METHOD

METHOD HaltEx 									: BOOL
END_METHOD

METHOD Jog 										: REFERENCE TO Tc2_MC2.ST_McOutputs
VAR_INPUT
	bFw											: BOOL;
	bBw											: BOOL;
END_VAR
END_METHOD

METHOD JogBwEx 									: BOOL
END_METHOD

METHOD JogClear 								: BOOL
END_METHOD

METHOD JogContinous 							: REFERENCE TO Tc2_MC2.ST_McOutputs
VAR_INPUT
	bFw											: BOOL;
	bBw											: BOOL;
END_VAR
END_METHOD

METHOD JogFast 									: REFERENCE TO Tc2_MC2.ST_McOutputs
VAR_INPUT
	bFw											: BOOL;
	bBw											: BOOL;
END_VAR
END_METHOD

METHOD JogFwEx 									: BOOL
END_METHOD

METHOD JogInching 								: REFERENCE TO Tc2_MC2.ST_McOutputs
VAR_INPUT
	bFw											: BOOL;
	bBw											: BOOL;
END_VAR
END_METHOD

METHOD JogInchingModulo 						: REFERENCE TO Tc2_MC2.ST_McOutputs
VAR_INPUT
	bFw											: BOOL;
	bBw											: BOOL;
END_VAR
END_METHOD

METHOD JogSlow 									: REFERENCE TO Tc2_MC2.ST_McOutputs
VAR_INPUT
	bFw											: BOOL;
	bBw											: BOOL;
END_VAR
END_METHOD

METHOD LimitSwitchDisable 						: REFERENCE TO Tc2_MC2.ST_McOutputs
VAR_INPUT
	bExecute									: BOOL;
END_VAR
END_METHOD

METHOD LimitSwitchDisableMax 					: REFERENCE TO Tc2_MC2.ST_McOutputs
VAR_INPUT
	bExecute									: BOOL;
END_VAR
END_METHOD

METHOD LimitSwitchDisableMin 					: REFERENCE TO Tc2_MC2.ST_McOutputs
VAR_INPUT
	bExecute									: BOOL;
END_VAR
END_METHOD

METHOD LimitSwitchEnable 						: REFERENCE TO Tc2_MC2.ST_McOutputs
VAR_INPUT
	bExecute									: BOOL;
END_VAR
END_METHOD

METHOD LimitSwitchEnableMax 					: REFERENCE TO Tc2_MC2.ST_McOutputs
VAR_INPUT
	bExecute									: BOOL;
END_VAR
END_METHOD

METHOD LimitSwitchEnableMin 					: REFERENCE TO Tc2_MC2.ST_McOutputs
VAR_INPUT
	bExecute									: BOOL;
END_VAR
END_METHOD

METHOD LimitSwitchRead 							: REFERENCE TO Tc2_MC2.ST_McOutputs
VAR_INPUT
	bExecute									: BOOL;
END_VAR
END_METHOD

METHOD LimitSwitchWrite 						: REFERENCE TO Tc2_MC2.ST_McOutputs
VAR_INPUT
	bExecute									: BOOL;
END_VAR
END_METHOD

METHOD LimitSwitchWriteMax 						: REFERENCE TO Tc2_MC2.ST_McOutputs
VAR_INPUT
	bExecute									: BOOL;
END_VAR
END_METHOD

METHOD LimitSwitchWriteMin 						: REFERENCE TO Tc2_MC2.ST_McOutputs
VAR_INPUT
	bExecute									: BOOL;
END_VAR
END_METHOD

METHOD Manual 									: BOOL
VAR_INPUT
	stManual									: REFERENCE TO ST_AxisControlManual;
END_VAR
END_METHOD

METHOD MoveAbsolute 							: REFERENCE TO Tc2_MC2.ST_McOutputs
VAR_INPUT
	bExecute									: BOOL;
END_VAR
END_METHOD

METHOD MoveAbsolute2 							: REFERENCE TO Tc2_MC2.ST_McOutputs
VAR_INPUT
	bExecute									: BOOL;
END_VAR
END_METHOD

METHOD MoveAbsoluteClear 						: BOOL
END_METHOD

METHOD MoveAbsoluteClear2 						: BOOL
END_METHOD

METHOD MoveAbsoluteEx 							: BOOL
END_METHOD

METHOD MoveAbsoluteEx2 							: BOOL
END_METHOD

